// TIA Portal project "Pompe_4" (V15.1)

(* hardware
DEVICE "S71500/ET200MP station_1"  S7-1500 station
   slot 0: "Rail_0"  Rack  6ES7 590-1***0-0AA0
   slot 1: "PLC_1"  CPU 1513-1 PN  6ES7 513-1AL02-0AB0  V2.6
      slot 3: "CPU display_1"  6ES7591-1AA00-0AA0
DEVICE "HMI_1"  KTP900 Basic PN
   slot 0: "HMI_1"  KTP900 Basic PN  6AV2 123-2JB03-0AX0  15.1.0.0
   slot 1: "HMI_RT_1"  KTP900 Basic PN  6AV2 123-2JB03-0AX0  15.1.0.0
   slot 5: "HMI_1.IE_CP_1"  PROFINET Interface  15.0.1.0
      slot 1: "PROFINET Interface_1"  PROFINET Interface
         slot 1: "Port_1"  Port
*)

// ===== PLC "PLC_1"  CPU 1513-1 PN =====

VAR_GLOBAL   // PLC tag table "Default tag table"
   "Clock_Byte" AT %MB0 : Byte;
   "Clock_10Hz" AT %M0.0 : Bool;
   "Clock_5Hz" AT %M0.1 : Bool;
   "Clock_2.5Hz" AT %M0.2 : Bool;
   "Clock_2Hz" AT %M0.3 : Bool;
   "Clock_1.25Hz" AT %M0.4 : Bool;
   "Clock_1Hz" AT %M0.5 : Bool;
   "Clock_0.625Hz" AT %M0.6 : Bool;
   "Clock_0.5Hz" AT %M0.7 : Bool;
END_VAR

TYPE "typeLogEntry"
   STRUCT
      Timestamp : DTL;
      Level : Real;
      Mode : DInt;
      ESD_Active : Bool;
      Fault_Active : Bool;
   END_STRUCT;
END_TYPE

// folder: Alarme/Avarii

DATA_BLOCK "Alarme_DB"   // DB1
{ S7_Optimized_Access := 'TRUE' }
VERSION : 0.1
   VAR
      gather : Word;
      "array" : Array[0..15] of Bool;
   END_VAR
BEGIN
END_DATA_BLOCK

DATA_BLOCK "Avarii_DB"   // DB2
{ S7_Optimized_Access := 'TRUE' }
VERSION : 0.1
   VAR
      esd_1 : Bool;
      btn_esd_1 : Bool;
      reset_esd_1 : Bool;
      avarie_sistem_1 : Bool;
      btn_avarie_sistem_1 : Bool;
      reset_avarie_sistem_1 : Bool;
      esd_2 : Bool;
      btn_esd_2 : Bool;
      reset_esd_2 : Bool;
      avarie_sistem_2 : Bool;
      btn_avarie_sistem_2 : Bool;
      reset_avarie_sistem_2 : Bool;
      esd_3 : Bool;
      btn_esd_3 : Bool;
      reset_esd_3 : Bool;
      avarie_sistem_3 : Bool;
      btn_avarie_sistem_3 : Bool;
      reset_avarie_sistem_3 : Bool;
      esd_4 : Bool;
      btn_esd_4 : Bool;
      reset_esd_4 : Bool;
      avarie_sistem_4 : Bool;
      btn_avarie_sistem_4 : Bool;
      reset_avarie_sistem_4 : Bool;
   END_VAR
BEGIN
END_DATA_BLOCK

// folder: DB-Functii-Networks

DATA_BLOCK "Sistem_2"   // DB13
{ S7_Optimized_Access := 'TRUE' }
VERSION : 0.1
// stored: InstanceOfName Sistem
"Sistem"
BEGIN
END_DATA_BLOCK

DATA_BLOCK "Sistem_1"   // DB15
{ S7_Optimized_Access := 'TRUE' }
VERSION : 0.1
// stored: InstanceOfName Sistem
"Sistem"
BEGIN
END_DATA_BLOCK

DATA_BLOCK "Sistem_3"   // DB16
{ S7_Optimized_Access := 'TRUE' }
VERSION : 0.1
// stored: InstanceOfName Sistem
"Sistem"
BEGIN
END_DATA_BLOCK

DATA_BLOCK "Sistem_4"   // DB17
{ S7_Optimized_Access := 'TRUE' }
VERSION : 0.1
// stored: InstanceOfName Sistem
"Sistem"
BEGIN
END_DATA_BLOCK

DATA_BLOCK "Logs_DB_1"   // DB21
{ S7_Optimized_Access := 'TRUE' }
VERSION : 0.1
// stored: InstanceOfName Logs
"Logs"
BEGIN
END_DATA_BLOCK

DATA_BLOCK "Logs_DB_2"   // DB22
{ S7_Optimized_Access := 'TRUE' }
VERSION : 0.1
// stored: InstanceOfName Logs
"Logs"
BEGIN
END_DATA_BLOCK

DATA_BLOCK "Logs_DB_3"   // DB23
{ S7_Optimized_Access := 'TRUE' }
VERSION : 0.1
// stored: InstanceOfName Logs
"Logs"
BEGIN
END_DATA_BLOCK

DATA_BLOCK "Logs_DB_4"   // DB24
{ S7_Optimized_Access := 'TRUE' }
VERSION : 0.1
// stored: InstanceOfName Logs
"Logs"
BEGIN
END_DATA_BLOCK

// folder: DB-Functii-Networks/DB-Functii-Sistem

DATA_BLOCK "Pompa_sistem_1"   // DB8
{ S7_Optimized_Access := 'TRUE' }
VERSION : 0.1
// stored: InstanceOfName Pompa
"Pompa"
BEGIN
END_DATA_BLOCK

DATA_BLOCK "Vana_sistem_1"   // DB9
{ S7_Optimized_Access := 'TRUE' }
VERSION : 0.1
// stored: InstanceOfName Vana
"Vana"
BEGIN
END_DATA_BLOCK

DATA_BLOCK "Simulare_sistem_1"   // DB14
{ S7_Optimized_Access := 'TRUE' }
VERSION : 0.1
// stored: InstanceOfName Simulare
"Simulare"
BEGIN
END_DATA_BLOCK

// folder: Logs

DATA_BLOCK "Logs1_DB"   // DB7
{ S7_Optimized_Access := 'TRUE' }
VERSION : 0.1
   VAR
      Log_Array : Array[0..100] of "typeLogEntry";
      index : Int;
      index_write : Int;
      target_index : Int;
      btn_jump : Bool;
      btn_prev : Bool;
      btn_next : Bool;
      btn_latest : Bool;
      Display_Entry : "typeLogEntry";
   END_VAR
BEGIN
END_DATA_BLOCK

DATA_BLOCK "Logs2_DB"   // DB25
{ S7_Optimized_Access := 'TRUE' }
VERSION : 0.1
   VAR
      Log_Array : Array[0..100] of "typeLogEntry";
      index : Int;
      index_write : Int;
      target_index : Int;
      btn_jump : Bool;
      btn_prev : Bool;
      btn_next : Bool;
      btn_latest : Bool;
      Display_Entry : "typeLogEntry";
   END_VAR
BEGIN
END_DATA_BLOCK

DATA_BLOCK "Logs3_DB"   // DB26
{ S7_Optimized_Access := 'TRUE' }
VERSION : 0.1
   VAR
      Log_Array : Array[0..100] of "typeLogEntry";
      index : Int;
      index_write : Int;
      target_index : Int;
      btn_jump : Bool;
      btn_prev : Bool;
      btn_next : Bool;
      btn_latest : Bool;
      Display_Entry : "typeLogEntry";
   END_VAR
BEGIN
END_DATA_BLOCK

DATA_BLOCK "Logs4_DB"   // DB27
{ S7_Optimized_Access := 'TRUE' }
VERSION : 0.1
   VAR
      Log_Array : Array[0..100] of "typeLogEntry";
      index : Int;
      index_write : Int;
      target_index : Int;
      btn_jump : Bool;
      btn_prev : Bool;
      btn_next : Bool;
      btn_latest : Bool;
      Display_Entry : "typeLogEntry";
   END_VAR
BEGIN
END_DATA_BLOCK

// folder: Sisteme_DB

DATA_BLOCK "Sistem_1_DB"   // DB3
{ S7_Optimized_Access := 'TRUE' }
VERSION : 0.1
   VAR
      nivel_maxim : Real := 100.0;
      debit_vana : Real := 2.5;
      debit_pompa : Real := 2.5;
      comanda_pornire_pompa : Bool;
      comanda_pornire_vana : Bool;
      pornire_pompa_pid : Bool;
      pornire_vana_pid : Bool;
      permisiune_start : Bool;
      setpoint_pid : Real;
      nivel_bazin : Real;
      pid_output : Real;
      btn_start : Bool;
      btn_stop : Bool;
      plecare_pompa : Bool;
      plecare_vana : Bool;
      indicator_pornit : Bool;
      "mod" : DInt;
   END_VAR
BEGIN
END_DATA_BLOCK

DATA_BLOCK "Sistem_2_DB"   // DB4
{ S7_Optimized_Access := 'TRUE' }
VERSION : 0.1
   VAR
      nivel_maxim : Real := 100.0;
      debit_vana : Real := 3.4;
      debit_pompa : Real := 1.3;
      comanda_pornire_pompa : Bool;
      comanda_pornire_vana : Bool;
      pornire_pompa_pid : Bool;
      pornire_vana_pid : Bool;
      permisiune_start : Bool;
      setpoint_pid : Real;
      nivel_bazin : Real;
      pid_output : Real;
      btn_start : Bool;
      btn_stop : Bool;
      plecare_pompa : Bool;
      plecare_vana : Bool;
      indicator_pornit : Bool;
      "mod" : DInt;
   END_VAR
BEGIN
END_DATA_BLOCK

DATA_BLOCK "Sistem_3_DB"   // DB5
{ S7_Optimized_Access := 'TRUE' }
VERSION : 0.1
   VAR
      nivel_maxim : Real := 100.0;
      debit_vana : Real := 5.7;
      debit_pompa : Real := 1.2;
      comanda_pornire_pompa : Bool;
      comanda_pornire_vana : Bool;
      pornire_pompa_pid : Bool;
      pornire_vana_pid : Bool;
      permisiune_start : Bool;
      setpoint_pid : Real;
      nivel_bazin : Real;
      pid_output : Real;
      btn_start : Bool;
      btn_stop : Bool;
      plecare_pompa : Bool;
      plecare_vana : Bool;
      indicator_pornit : Bool;
      "mod" : DInt;
   END_VAR
BEGIN
END_DATA_BLOCK

DATA_BLOCK "Sistem_4_DB"   // DB6
{ S7_Optimized_Access := 'TRUE' }
VERSION : 0.1
   VAR
      nivel_maxim : Real := 100.0;
      debit_vana : Real := 1.8;
      debit_pompa : Real := 3.6;
      comanda_pornire_pompa : Bool;
      comanda_pornire_vana : Bool;
      pornire_pompa_pid : Bool;
      pornire_vana_pid : Bool;
      permisiune_start : Bool;
      setpoint_pid : Real;
      nivel_bazin : Real;
      pid_output : Real;
      btn_start : Bool;
      btn_stop : Bool;
      plecare_pompa : Bool;
      plecare_vana : Bool;
      indicator_pornit : Bool;
      "mod" : DInt;
   END_VAR
BEGIN
END_DATA_BLOCK

// folder: System blocks/Program resources

DATA_BLOCK "timer_reset_pornire_vana"   // DB10
{ S7_Optimized_Access := 'TRUE' }
AUTHOR : Simatic
FAMILY : IEC
NAME : IEC_TMR
VERSION : 1.0
// stored: InstanceOfName IEC_TIMER
"IEC_TIMER"
BEGIN
END_DATA_BLOCK

DATA_BLOCK "timer_reset_pornire_pompa"   // DB11
{ S7_Optimized_Access := 'TRUE' }
AUTHOR : Simatic
FAMILY : IEC
NAME : IEC_TMR
VERSION : 1.0
// stored: InstanceOfName IEC_TIMER
"IEC_TIMER"
BEGIN
END_DATA_BLOCK

// folder: (top level)

ORGANIZATION_BLOCK "Main"   // OB1, LAD, ProgramCycle
TITLE = "Main Program Sweep (Cycle)"
{ S7_Optimized_Access := 'TRUE' }
VERSION : 0.1
   VAR_INPUT
      Initial_Call : Bool;   // Initial call of this OB
      Remanence : Bool;   // =True, if remanent data are available
   END_VAR
BEGIN

REGION Network 1: Gather pe alarme
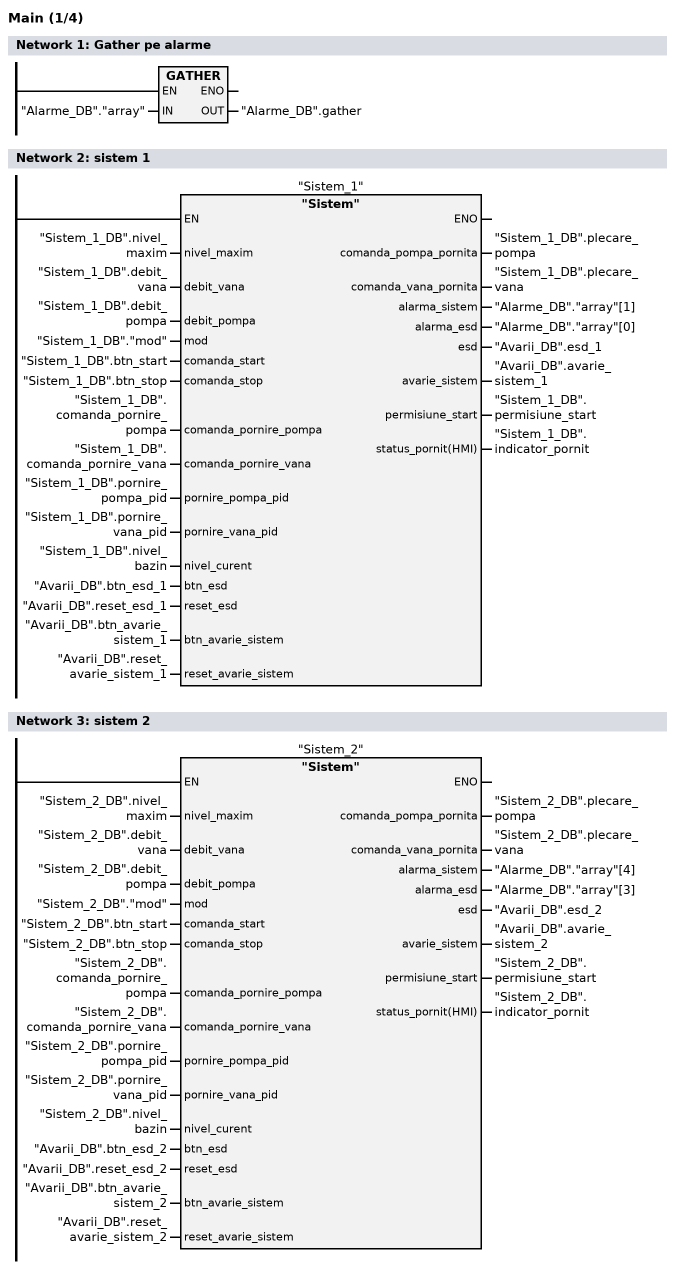
   GATHER(IN := "Alarme_DB"."array", OUT => "Alarme_DB".gather);
END_REGION

REGION Network 2: sistem 1
   RUNG wire#powerrail
      "Sistem_1"(nivel_maxim := "Sistem_1_DB".nivel_maxim, debit_vana := "Sistem_1_DB".debit_vana, debit_pompa := "Sistem_1_DB".debit_pompa, "mod" := "Sistem_1_DB"."mod", comanda_start := "Sistem_1_DB".btn_start, comanda_stop := "Sistem_1_DB".btn_stop, comanda_pornire_pompa := "Sistem_1_DB".comanda_pornire_pompa, comanda_pornire_vana := "Sistem_1_DB".comanda_pornire_vana, pornire_pompa_pid := "Sistem_1_DB".pornire_pompa_pid, pornire_vana_pid := "Sistem_1_DB".pornire_vana_pid, nivel_curent := "Sistem_1_DB".nivel_bazin, btn_esd := "Avarii_DB".btn_esd_1, reset_esd := "Avarii_DB".reset_esd_1, btn_avarie_sistem := "Avarii_DB".btn_avarie_sistem_1, reset_avarie_sistem := "Avarii_DB".reset_avarie_sistem_1, comanda_pompa_pornita => "Sistem_1_DB".plecare_pompa, comanda_vana_pornita => "Sistem_1_DB".plecare_vana, alarma_sistem => "Alarme_DB"."array"[1], alarma_esd => "Alarme_DB"."array"[0], esd => "Avarii_DB".esd_1, avarie_sistem => "Avarii_DB".avarie_sistem_1, permisiune_start => "Sistem_1_DB".permisiune_start, "status_pornit(HMI)" => "Sistem_1_DB".indicator_pornit)
   END_RUNG
   // the same network as SCL:
   "Sistem_1"(nivel_maxim := "Sistem_1_DB".nivel_maxim,   // "Sistem"
              debit_vana := "Sistem_1_DB".debit_vana,
              debit_pompa := "Sistem_1_DB".debit_pompa,
              "mod" := "Sistem_1_DB"."mod",
              comanda_start := "Sistem_1_DB".btn_start,
              comanda_stop := "Sistem_1_DB".btn_stop,
              comanda_pornire_pompa := "Sistem_1_DB".comanda_pornire_pompa,
              comanda_pornire_vana := "Sistem_1_DB".comanda_pornire_vana,
              pornire_pompa_pid := "Sistem_1_DB".pornire_pompa_pid,
              pornire_vana_pid := "Sistem_1_DB".pornire_vana_pid,
              nivel_curent := "Sistem_1_DB".nivel_bazin,
              btn_esd := "Avarii_DB".btn_esd_1,
              reset_esd := "Avarii_DB".reset_esd_1,
              btn_avarie_sistem := "Avarii_DB".btn_avarie_sistem_1,
              reset_avarie_sistem := "Avarii_DB".reset_avarie_sistem_1,
              comanda_pompa_pornita => "Sistem_1_DB".plecare_pompa,
              comanda_vana_pornita => "Sistem_1_DB".plecare_vana,
              alarma_sistem => "Alarme_DB"."array"[1],
              alarma_esd => "Alarme_DB"."array"[0],
              esd => "Avarii_DB".esd_1,
              avarie_sistem => "Avarii_DB".avarie_sistem_1,
              permisiune_start => "Sistem_1_DB".permisiune_start,
              "status_pornit(HMI)" => "Sistem_1_DB".indicator_pornit);
END_REGION

REGION Network 3: sistem 2
   RUNG wire#powerrail
      "Sistem_2"(nivel_maxim := "Sistem_2_DB".nivel_maxim, debit_vana := "Sistem_2_DB".debit_vana, debit_pompa := "Sistem_2_DB".debit_pompa, "mod" := "Sistem_2_DB"."mod", comanda_start := "Sistem_2_DB".btn_start, comanda_stop := "Sistem_2_DB".btn_stop, comanda_pornire_pompa := "Sistem_2_DB".comanda_pornire_pompa, comanda_pornire_vana := "Sistem_2_DB".comanda_pornire_vana, pornire_pompa_pid := "Sistem_2_DB".pornire_pompa_pid, pornire_vana_pid := "Sistem_2_DB".pornire_vana_pid, nivel_curent := "Sistem_2_DB".nivel_bazin, btn_esd := "Avarii_DB".btn_esd_2, reset_esd := "Avarii_DB".reset_esd_2, btn_avarie_sistem := "Avarii_DB".btn_avarie_sistem_2, reset_avarie_sistem := "Avarii_DB".reset_avarie_sistem_2, comanda_pompa_pornita => "Sistem_2_DB".plecare_pompa, comanda_vana_pornita => "Sistem_2_DB".plecare_vana, alarma_sistem => "Alarme_DB"."array"[4], alarma_esd => "Alarme_DB"."array"[3], esd => "Avarii_DB".esd_2, avarie_sistem => "Avarii_DB".avarie_sistem_2, permisiune_start => "Sistem_2_DB".permisiune_start, "status_pornit(HMI)" => "Sistem_2_DB".indicator_pornit)
   END_RUNG
   // the same network as SCL:
   "Sistem_2"(nivel_maxim := "Sistem_2_DB".nivel_maxim,   // "Sistem"
              debit_vana := "Sistem_2_DB".debit_vana,
              debit_pompa := "Sistem_2_DB".debit_pompa,
              "mod" := "Sistem_2_DB"."mod",
              comanda_start := "Sistem_2_DB".btn_start,
              comanda_stop := "Sistem_2_DB".btn_stop,
              comanda_pornire_pompa := "Sistem_2_DB".comanda_pornire_pompa,
              comanda_pornire_vana := "Sistem_2_DB".comanda_pornire_vana,
              pornire_pompa_pid := "Sistem_2_DB".pornire_pompa_pid,
              pornire_vana_pid := "Sistem_2_DB".pornire_vana_pid,
              nivel_curent := "Sistem_2_DB".nivel_bazin,
              btn_esd := "Avarii_DB".btn_esd_2,
              reset_esd := "Avarii_DB".reset_esd_2,
              btn_avarie_sistem := "Avarii_DB".btn_avarie_sistem_2,
              reset_avarie_sistem := "Avarii_DB".reset_avarie_sistem_2,
              comanda_pompa_pornita => "Sistem_2_DB".plecare_pompa,
              comanda_vana_pornita => "Sistem_2_DB".plecare_vana,
              alarma_sistem => "Alarme_DB"."array"[4],
              alarma_esd => "Alarme_DB"."array"[3],
              esd => "Avarii_DB".esd_2,
              avarie_sistem => "Avarii_DB".avarie_sistem_2,
              permisiune_start => "Sistem_2_DB".permisiune_start,
              "status_pornit(HMI)" => "Sistem_2_DB".indicator_pornit);
END_REGION

REGION Network 4: sistem 3
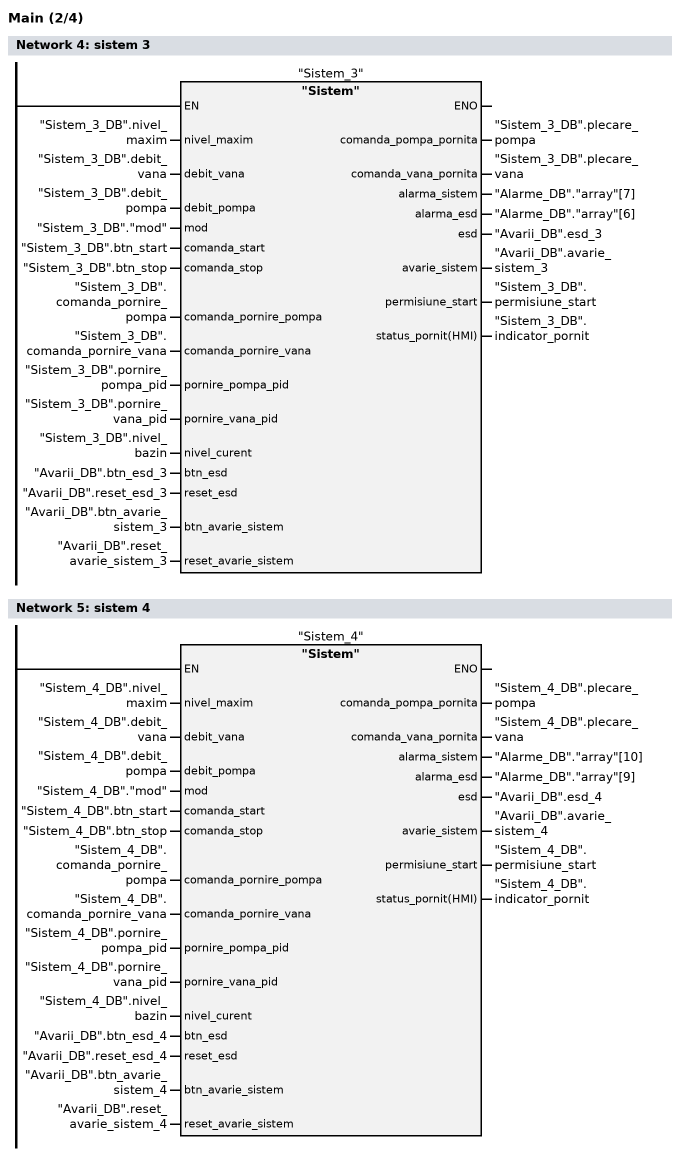
   RUNG wire#powerrail
      "Sistem_3"(nivel_maxim := "Sistem_3_DB".nivel_maxim, debit_vana := "Sistem_3_DB".debit_vana, debit_pompa := "Sistem_3_DB".debit_pompa, "mod" := "Sistem_3_DB"."mod", comanda_start := "Sistem_3_DB".btn_start, comanda_stop := "Sistem_3_DB".btn_stop, comanda_pornire_pompa := "Sistem_3_DB".comanda_pornire_pompa, comanda_pornire_vana := "Sistem_3_DB".comanda_pornire_vana, pornire_pompa_pid := "Sistem_3_DB".pornire_pompa_pid, pornire_vana_pid := "Sistem_3_DB".pornire_vana_pid, nivel_curent := "Sistem_3_DB".nivel_bazin, btn_esd := "Avarii_DB".btn_esd_3, reset_esd := "Avarii_DB".reset_esd_3, btn_avarie_sistem := "Avarii_DB".btn_avarie_sistem_3, reset_avarie_sistem := "Avarii_DB".reset_avarie_sistem_3, comanda_pompa_pornita => "Sistem_3_DB".plecare_pompa, comanda_vana_pornita => "Sistem_3_DB".plecare_vana, alarma_sistem => "Alarme_DB"."array"[7], alarma_esd => "Alarme_DB"."array"[6], esd => "Avarii_DB".esd_3, avarie_sistem => "Avarii_DB".avarie_sistem_3, permisiune_start => "Sistem_3_DB".permisiune_start, "status_pornit(HMI)" => "Sistem_3_DB".indicator_pornit)
   END_RUNG
   // the same network as SCL:
   "Sistem_3"(nivel_maxim := "Sistem_3_DB".nivel_maxim,   // "Sistem"
              debit_vana := "Sistem_3_DB".debit_vana,
              debit_pompa := "Sistem_3_DB".debit_pompa,
              "mod" := "Sistem_3_DB"."mod",
              comanda_start := "Sistem_3_DB".btn_start,
              comanda_stop := "Sistem_3_DB".btn_stop,
              comanda_pornire_pompa := "Sistem_3_DB".comanda_pornire_pompa,
              comanda_pornire_vana := "Sistem_3_DB".comanda_pornire_vana,
              pornire_pompa_pid := "Sistem_3_DB".pornire_pompa_pid,
              pornire_vana_pid := "Sistem_3_DB".pornire_vana_pid,
              nivel_curent := "Sistem_3_DB".nivel_bazin,
              btn_esd := "Avarii_DB".btn_esd_3,
              reset_esd := "Avarii_DB".reset_esd_3,
              btn_avarie_sistem := "Avarii_DB".btn_avarie_sistem_3,
              reset_avarie_sistem := "Avarii_DB".reset_avarie_sistem_3,
              comanda_pompa_pornita => "Sistem_3_DB".plecare_pompa,
              comanda_vana_pornita => "Sistem_3_DB".plecare_vana,
              alarma_sistem => "Alarme_DB"."array"[7],
              alarma_esd => "Alarme_DB"."array"[6],
              esd => "Avarii_DB".esd_3,
              avarie_sistem => "Avarii_DB".avarie_sistem_3,
              permisiune_start => "Sistem_3_DB".permisiune_start,
              "status_pornit(HMI)" => "Sistem_3_DB".indicator_pornit);
END_REGION

REGION Network 5: sistem 4
   RUNG wire#powerrail
      "Sistem_4"(nivel_maxim := "Sistem_4_DB".nivel_maxim, debit_vana := "Sistem_4_DB".debit_vana, debit_pompa := "Sistem_4_DB".debit_pompa, "mod" := "Sistem_4_DB"."mod", comanda_start := "Sistem_4_DB".btn_start, comanda_stop := "Sistem_4_DB".btn_stop, comanda_pornire_pompa := "Sistem_4_DB".comanda_pornire_pompa, comanda_pornire_vana := "Sistem_4_DB".comanda_pornire_vana, pornire_pompa_pid := "Sistem_4_DB".pornire_pompa_pid, pornire_vana_pid := "Sistem_4_DB".pornire_vana_pid, nivel_curent := "Sistem_4_DB".nivel_bazin, btn_esd := "Avarii_DB".btn_esd_4, reset_esd := "Avarii_DB".reset_esd_4, btn_avarie_sistem := "Avarii_DB".btn_avarie_sistem_4, reset_avarie_sistem := "Avarii_DB".reset_avarie_sistem_4, comanda_pompa_pornita => "Sistem_4_DB".plecare_pompa, comanda_vana_pornita => "Sistem_4_DB".plecare_vana, alarma_sistem => "Alarme_DB"."array"[10], alarma_esd => "Alarme_DB"."array"[9], esd => "Avarii_DB".esd_4, avarie_sistem => "Avarii_DB".avarie_sistem_4, permisiune_start => "Sistem_4_DB".permisiune_start, "status_pornit(HMI)" => "Sistem_4_DB".indicator_pornit)
   END_RUNG
   // the same network as SCL:
   "Sistem_4"(nivel_maxim := "Sistem_4_DB".nivel_maxim,   // "Sistem"
              debit_vana := "Sistem_4_DB".debit_vana,
              debit_pompa := "Sistem_4_DB".debit_pompa,
              "mod" := "Sistem_4_DB"."mod",
              comanda_start := "Sistem_4_DB".btn_start,
              comanda_stop := "Sistem_4_DB".btn_stop,
              comanda_pornire_pompa := "Sistem_4_DB".comanda_pornire_pompa,
              comanda_pornire_vana := "Sistem_4_DB".comanda_pornire_vana,
              pornire_pompa_pid := "Sistem_4_DB".pornire_pompa_pid,
              pornire_vana_pid := "Sistem_4_DB".pornire_vana_pid,
              nivel_curent := "Sistem_4_DB".nivel_bazin,
              btn_esd := "Avarii_DB".btn_esd_4,
              reset_esd := "Avarii_DB".reset_esd_4,
              btn_avarie_sistem := "Avarii_DB".btn_avarie_sistem_4,
              reset_avarie_sistem := "Avarii_DB".reset_avarie_sistem_4,
              comanda_pompa_pornita => "Sistem_4_DB".plecare_pompa,
              comanda_vana_pornita => "Sistem_4_DB".plecare_vana,
              alarma_sistem => "Alarme_DB"."array"[10],
              alarma_esd => "Alarme_DB"."array"[9],
              esd => "Avarii_DB".esd_4,
              avarie_sistem => "Avarii_DB".avarie_sistem_4,
              permisiune_start => "Sistem_4_DB".permisiune_start,
              "status_pornit(HMI)" => "Sistem_4_DB".indicator_pornit);
END_REGION

REGION Network 6: logs 1
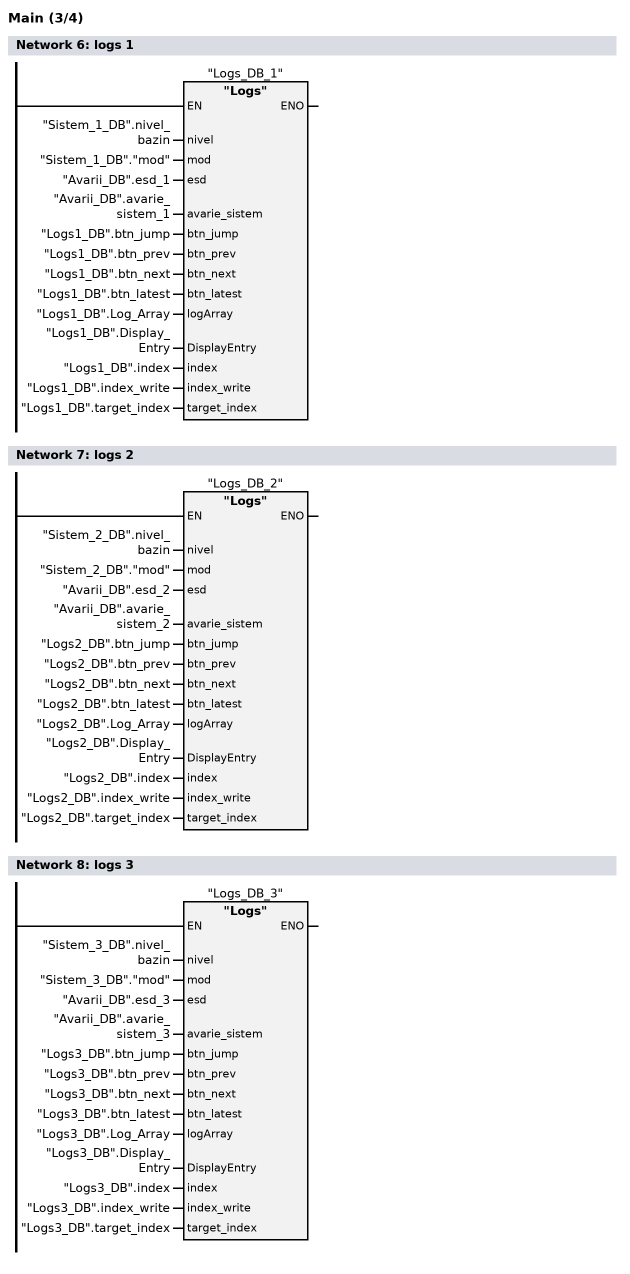
   RUNG wire#powerrail
      "Logs_DB_1"(nivel := "Sistem_1_DB".nivel_bazin, "mod" := "Sistem_1_DB"."mod", esd := "Avarii_DB".esd_1, avarie_sistem := "Avarii_DB".avarie_sistem_1, btn_jump := "Logs1_DB".btn_jump, btn_prev := "Logs1_DB".btn_prev, btn_next := "Logs1_DB".btn_next, btn_latest := "Logs1_DB".btn_latest, logArray := "Logs1_DB".Log_Array, DisplayEntry := "Logs1_DB".Display_Entry, index := "Logs1_DB".index, index_write := "Logs1_DB".index_write, target_index := "Logs1_DB".target_index)
   END_RUNG
   // the same network as SCL:
   "Logs_DB_1"(nivel := "Sistem_1_DB".nivel_bazin,   // "Logs"
               "mod" := "Sistem_1_DB"."mod",
               esd := "Avarii_DB".esd_1,
               avarie_sistem := "Avarii_DB".avarie_sistem_1,
               btn_jump := "Logs1_DB".btn_jump,
               btn_prev := "Logs1_DB".btn_prev,
               btn_next := "Logs1_DB".btn_next,
               btn_latest := "Logs1_DB".btn_latest,
               logArray := "Logs1_DB".Log_Array,
               DisplayEntry := "Logs1_DB".Display_Entry,
               index := "Logs1_DB".index,
               index_write := "Logs1_DB".index_write,
               target_index := "Logs1_DB".target_index);
END_REGION

REGION Network 7: logs 2
   RUNG wire#powerrail
      "Logs_DB_2"(nivel := "Sistem_2_DB".nivel_bazin, "mod" := "Sistem_2_DB"."mod", esd := "Avarii_DB".esd_2, avarie_sistem := "Avarii_DB".avarie_sistem_2, btn_jump := "Logs2_DB".btn_jump, btn_prev := "Logs2_DB".btn_prev, btn_next := "Logs2_DB".btn_next, btn_latest := "Logs2_DB".btn_latest, logArray := "Logs2_DB".Log_Array, DisplayEntry := "Logs2_DB".Display_Entry, index := "Logs2_DB".index, index_write := "Logs2_DB".index_write, target_index := "Logs2_DB".target_index)
   END_RUNG
   // the same network as SCL:
   "Logs_DB_2"(nivel := "Sistem_2_DB".nivel_bazin,   // "Logs"
               "mod" := "Sistem_2_DB"."mod",
               esd := "Avarii_DB".esd_2,
               avarie_sistem := "Avarii_DB".avarie_sistem_2,
               btn_jump := "Logs2_DB".btn_jump,
               btn_prev := "Logs2_DB".btn_prev,
               btn_next := "Logs2_DB".btn_next,
               btn_latest := "Logs2_DB".btn_latest,
               logArray := "Logs2_DB".Log_Array,
               DisplayEntry := "Logs2_DB".Display_Entry,
               index := "Logs2_DB".index,
               index_write := "Logs2_DB".index_write,
               target_index := "Logs2_DB".target_index);
END_REGION

REGION Network 8: logs 3
   RUNG wire#powerrail
      "Logs_DB_3"(nivel := "Sistem_3_DB".nivel_bazin, "mod" := "Sistem_3_DB"."mod", esd := "Avarii_DB".esd_3, avarie_sistem := "Avarii_DB".avarie_sistem_3, btn_jump := "Logs3_DB".btn_jump, btn_prev := "Logs3_DB".btn_prev, btn_next := "Logs3_DB".btn_next, btn_latest := "Logs3_DB".btn_latest, logArray := "Logs3_DB".Log_Array, DisplayEntry := "Logs3_DB".Display_Entry, index := "Logs3_DB".index, index_write := "Logs3_DB".index_write, target_index := "Logs3_DB".target_index)
   END_RUNG
   // the same network as SCL:
   "Logs_DB_3"(nivel := "Sistem_3_DB".nivel_bazin,   // "Logs"
               "mod" := "Sistem_3_DB"."mod",
               esd := "Avarii_DB".esd_3,
               avarie_sistem := "Avarii_DB".avarie_sistem_3,
               btn_jump := "Logs3_DB".btn_jump,
               btn_prev := "Logs3_DB".btn_prev,
               btn_next := "Logs3_DB".btn_next,
               btn_latest := "Logs3_DB".btn_latest,
               logArray := "Logs3_DB".Log_Array,
               DisplayEntry := "Logs3_DB".Display_Entry,
               index := "Logs3_DB".index,
               index_write := "Logs3_DB".index_write,
               target_index := "Logs3_DB".target_index);
END_REGION

REGION Network 9: logs 4
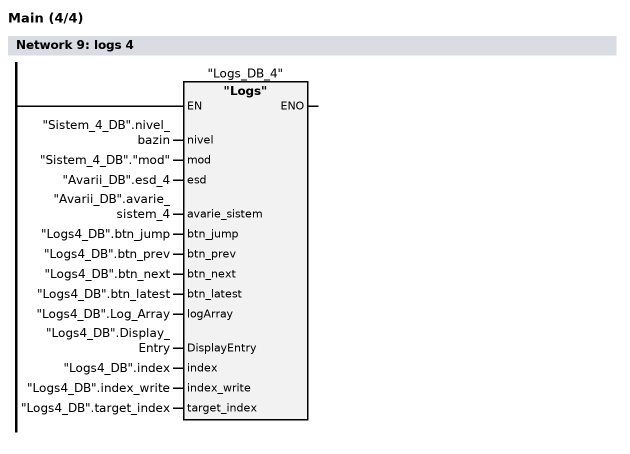
   RUNG wire#powerrail
      "Logs_DB_4"(nivel := "Sistem_4_DB".nivel_bazin, "mod" := "Sistem_4_DB"."mod", esd := "Avarii_DB".esd_4, avarie_sistem := "Avarii_DB".avarie_sistem_4, btn_jump := "Logs4_DB".btn_jump, btn_prev := "Logs4_DB".btn_prev, btn_next := "Logs4_DB".btn_next, btn_latest := "Logs4_DB".btn_latest, logArray := "Logs4_DB".Log_Array, DisplayEntry := "Logs4_DB".Display_Entry, index := "Logs4_DB".index, index_write := "Logs4_DB".index_write, target_index := "Logs4_DB".target_index)
   END_RUNG
   // the same network as SCL:
   "Logs_DB_4"(nivel := "Sistem_4_DB".nivel_bazin,   // "Logs"
               "mod" := "Sistem_4_DB"."mod",
               esd := "Avarii_DB".esd_4,
               avarie_sistem := "Avarii_DB".avarie_sistem_4,
               btn_jump := "Logs4_DB".btn_jump,
               btn_prev := "Logs4_DB".btn_prev,
               btn_next := "Logs4_DB".btn_next,
               btn_latest := "Logs4_DB".btn_latest,
               logArray := "Logs4_DB".Log_Array,
               DisplayEntry := "Logs4_DB".Display_Entry,
               index := "Logs4_DB".index,
               index_write := "Logs4_DB".index_write,
               target_index := "Logs4_DB".target_index);
END_REGION
END_ORGANIZATION_BLOCK

// folder: FB-Sistem

FUNCTION_BLOCK "Sistem"   // FB1, LAD
{ S7_Optimized_Access := 'TRUE' }
VERSION : 0.1
   VAR_INPUT
      nivel_maxim : Real;
      debit_vana : Real;
      debit_pompa : Real;
      "mod" : DInt;
   END_VAR
   VAR_OUTPUT
      comanda_pompa_pornita : Bool;
      comanda_vana_pornita : Bool;
      alarma_sistem : Bool;
      alarma_esd : Bool;
      esd : Bool;
      avarie_sistem : Bool;
      permisiune_start : Bool;
      "status_pornit(HMI)" : Bool;
   END_VAR
   VAR_IN_OUT
      comanda_start : Bool;
      comanda_stop : Bool;
      comanda_pornire_pompa : Bool;
      comanda_pornire_vana : Bool;
      pornire_pompa_pid : Bool;
      pornire_vana_pid : Bool;
      nivel_curent : Real;
      btn_esd : Bool;
      reset_esd : Bool;
      btn_avarie_sistem : Bool;
      reset_avarie_sistem : Bool;
   END_VAR
   VAR
      status_pornit_pompa : Bool;
      status_pornit_vana : Bool;
      resetare_comanda_vana : Bool;
      resetare_comanda_pompa : Bool;
      timer_reset_esd : TON_TIME;
      timer_reset_avarie_sistem : TON_TIME;
      timer_reset_comanda_stop : TON_TIME;
      Simulare_Instance : "Simulare";
      Vana_Instance : "Vana";
      Pompa_Instance : "Pompa";
   END_VAR
   VAR_TEMP   // added for the SCL form of the ladder/FBD networks
      _w1 : Bool;
      _w2 : Bool;
   END_VAR
BEGIN

REGION Network 1: comanda buton start
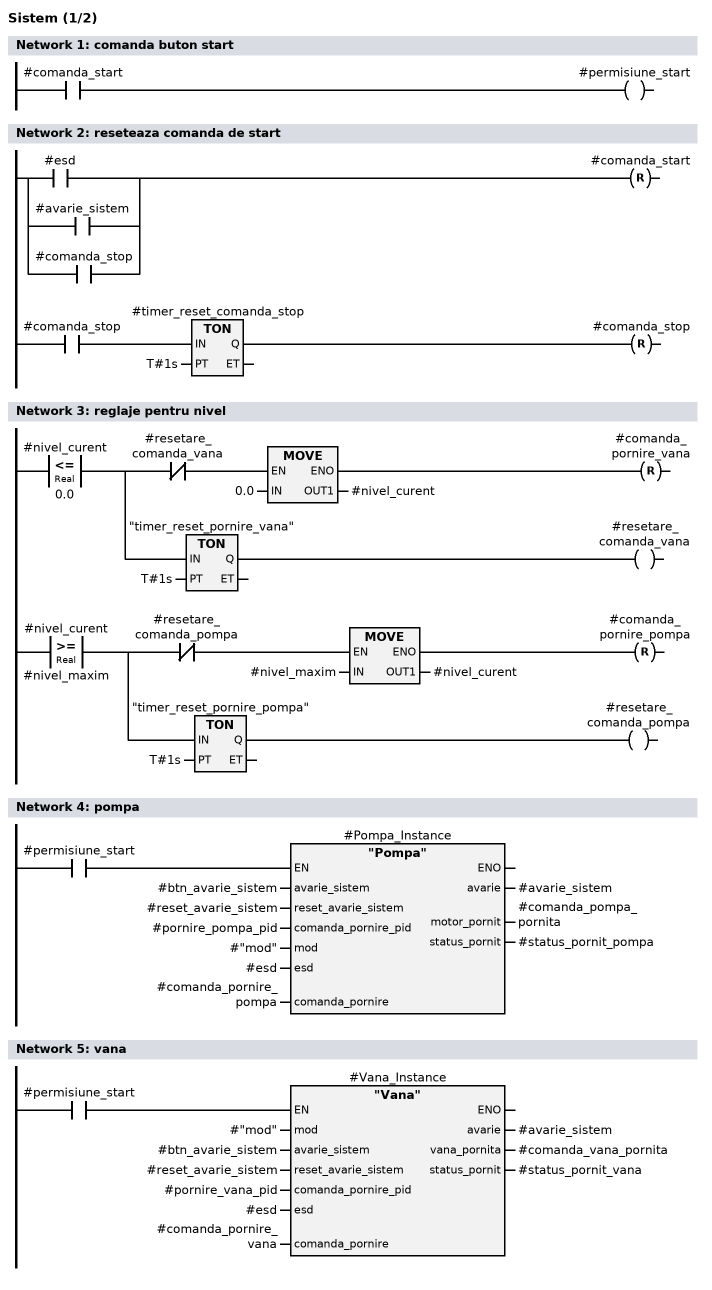
   RUNG wire#powerrail
      Contact( #comanda_start )
      Coil( #permisiune_start )
   END_RUNG
   // the same network as SCL:
   #permisiune_start := #comanda_start;
END_REGION

REGION Network 2: reseteaza comanda de start
   IF #esd OR #avarie_sistem OR #comanda_stop THEN #comanda_start := FALSE; END_IF;
   #timer_reset_comanda_stop(IN := #comanda_stop, PT := T#1s);   // TON
   IF #timer_reset_comanda_stop.Q THEN #comanda_stop := FALSE; END_IF;
END_REGION

REGION Network 3: reglaje pentru nivel
   #_w1 := #nivel_curent <= 0.0;
   IF #_w1 AND NOT #resetare_comanda_vana THEN
       #nivel_curent := 0.0;
       #comanda_pornire_vana := FALSE;
   END_IF;
   "timer_reset_pornire_vana".TON(IN := #_w1, PT := T#1s);
   #resetare_comanda_vana := "timer_reset_pornire_vana".Q;
   #_w2 := #nivel_curent >= #nivel_maxim;
   IF #_w2 AND NOT #resetare_comanda_pompa THEN
       #nivel_curent := #nivel_maxim;
       #comanda_pornire_pompa := FALSE;
   END_IF;
   "timer_reset_pornire_pompa".TON(IN := #_w2, PT := T#1s);
   #resetare_comanda_pompa := "timer_reset_pornire_pompa".Q;
END_REGION

REGION Network 4: pompa
   RUNG wire#powerrail
      Contact( #permisiune_start )
      #Pompa_Instance(avarie_sistem := #btn_avarie_sistem, reset_avarie_sistem := #reset_avarie_sistem, comanda_pornire_pid := #pornire_pompa_pid, "mod" := #"mod", esd := #esd, comanda_pornire := #comanda_pornire_pompa, avarie => #avarie_sistem, motor_pornit => #comanda_pompa_pornita, status_pornit => #status_pornit_pompa)
   END_RUNG
   // the same network as SCL:
   IF #permisiune_start THEN
       #Pompa_Instance(avarie_sistem := #btn_avarie_sistem,   // "Pompa"
                       reset_avarie_sistem := #reset_avarie_sistem,
                       comanda_pornire_pid := #pornire_pompa_pid,
                       "mod" := #"mod",
                       esd := #esd,
                       comanda_pornire := #comanda_pornire_pompa,
                       avarie => #avarie_sistem,
                       motor_pornit => #comanda_pompa_pornita,
                       status_pornit => #status_pornit_pompa);
   END_IF;
END_REGION

REGION Network 5: vana
   RUNG wire#powerrail
      Contact( #permisiune_start )
      #Vana_Instance("mod" := #"mod", avarie_sistem := #btn_avarie_sistem, reset_avarie_sistem := #reset_avarie_sistem, comanda_pornire_pid := #pornire_vana_pid, esd := #esd, comanda_pornire := #comanda_pornire_vana, avarie => #avarie_sistem, vana_pornita => #comanda_vana_pornita, status_pornit => #status_pornit_vana)
   END_RUNG
   // the same network as SCL:
   IF #permisiune_start THEN
       #Vana_Instance("mod" := #"mod",   // "Vana"
                      avarie_sistem := #btn_avarie_sistem,
                      reset_avarie_sistem := #reset_avarie_sistem,
                      comanda_pornire_pid := #pornire_vana_pid,
                      esd := #esd,
                      comanda_pornire := #comanda_pornire_vana,
                      avarie => #avarie_sistem,
                      vana_pornita => #comanda_vana_pornita,
                      status_pornit => #status_pornit_vana);
   END_IF;
END_REGION

REGION Network 6: status sistem pornit
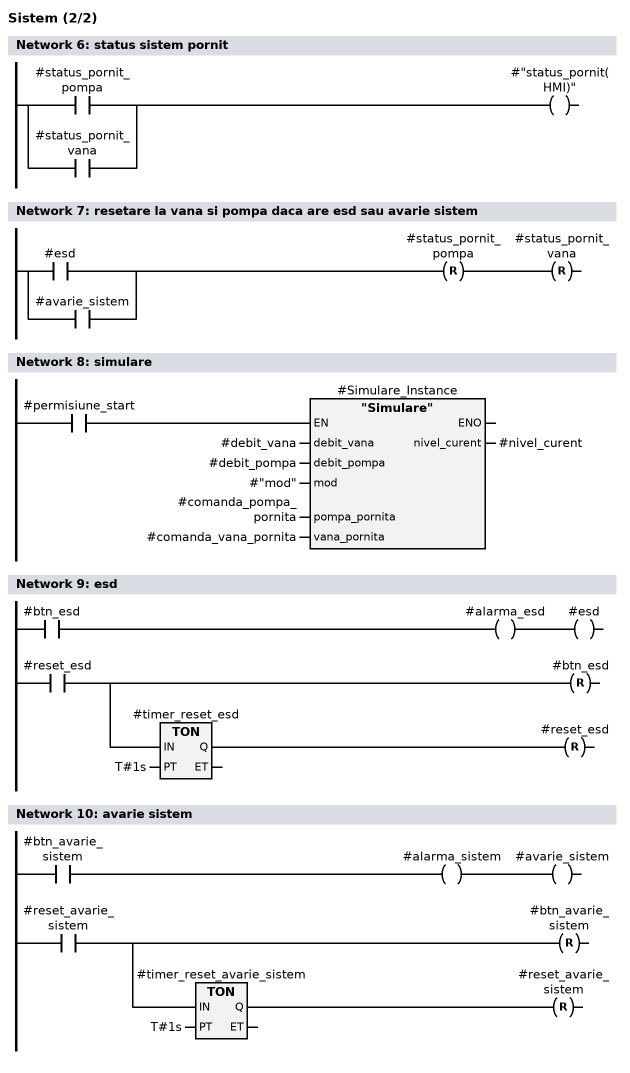
   RUNG wire#powerrail
      Contact( #status_pornit_pompa )
      wire#w1
      Coil( #"status_pornit(HMI)" )
   END_RUNG
   RUNG wire#powerrail
      Contact( #status_pornit_vana )
   END_RUNG wire#w1
   // the same network as SCL:
   #"status_pornit(HMI)" := #status_pornit_pompa OR #status_pornit_vana;
END_REGION

REGION Network 7: resetare la vana si pompa daca are esd sau avarie sistem
   RUNG wire#powerrail
      Contact( #esd )
      wire#w1
      R_Coil( #status_pornit_pompa )
      R_Coil( #status_pornit_vana )
   END_RUNG
   RUNG wire#powerrail
      Contact( #avarie_sistem )
   END_RUNG wire#w1
   // the same network as SCL:
   IF #esd OR #avarie_sistem THEN
       #status_pornit_pompa := FALSE;
       #status_pornit_vana := FALSE;
   END_IF;
END_REGION

REGION Network 8: simulare
   RUNG wire#powerrail
      Contact( #permisiune_start )
      #Simulare_Instance(debit_vana := #debit_vana, debit_pompa := #debit_pompa, "mod" := #"mod", pompa_pornita := #comanda_pompa_pornita, vana_pornita := #comanda_vana_pornita, nivel_curent => #nivel_curent)
   END_RUNG
   // the same network as SCL:
   IF #permisiune_start THEN
       #Simulare_Instance(debit_vana := #debit_vana,   // "Simulare"
                          debit_pompa := #debit_pompa,
                          "mod" := #"mod",
                          pompa_pornita := #comanda_pompa_pornita,
                          vana_pornita := #comanda_vana_pornita,
                          nivel_curent => #nivel_curent);
   END_IF;
END_REGION

REGION Network 9: esd
   #alarma_esd := #btn_esd;
   #esd := #btn_esd;
   IF #reset_esd THEN #btn_esd := FALSE; END_IF;
   #timer_reset_esd(IN := #reset_esd, PT := T#1s);   // TON
   IF #timer_reset_esd.Q THEN #reset_esd := FALSE; END_IF;
END_REGION

REGION Network 10: avarie sistem
   #alarma_sistem := #btn_avarie_sistem;
   #avarie_sistem := #btn_avarie_sistem;
   IF #reset_avarie_sistem THEN #btn_avarie_sistem := FALSE; END_IF;
   #timer_reset_avarie_sistem(IN := #reset_avarie_sistem, PT := T#1s);   // TON
   IF #timer_reset_avarie_sistem.Q THEN #reset_avarie_sistem := FALSE; END_IF;
END_REGION
END_FUNCTION_BLOCK

FUNCTION_BLOCK "Pompa"   // FB2, LAD
{ S7_Optimized_Access := 'TRUE' }
VERSION : 0.1
   VAR_INPUT
      avarie_sistem : Bool;
      reset_avarie_sistem : Bool;
      comanda_pornire_pid : Bool;
      "mod" : DInt;
      esd : Bool;
   END_VAR
   VAR_OUTPUT
      avarie : Bool;
      motor_pornit : Bool;
      status_pornit : Bool;
   END_VAR
   VAR_IN_OUT
      comanda_pornire : Bool;
   END_VAR
BEGIN

REGION Network 1: pornire pompa pe oricem od de functionare
   // 0 - manual, 1 - auto
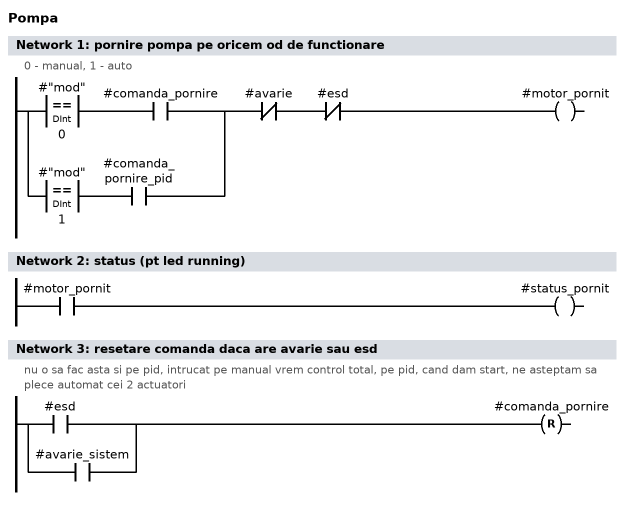
   RUNG wire#powerrail
      { S7_Templates := "SrcType := DInt" } EQ_Contact(in1 := #"mod", in2 := 0)
      Contact( #comanda_pornire )
      wire#w1
      I_Contact( #avarie )
      I_Contact( #esd )
      Coil( #motor_pornit )
   END_RUNG
   RUNG wire#powerrail
      { S7_Templates := "SrcType := DInt" } EQ_Contact(in1 := #"mod", in2 := 1)
      Contact( #comanda_pornire_pid )
   END_RUNG wire#w1
   // the same network as SCL:
   #motor_pornit := (((#"mod" = 0) AND #comanda_pornire) OR ((#"mod" = 1) AND #comanda_pornire_pid)) AND NOT #avarie AND NOT #esd;
END_REGION

REGION Network 2: status (pt led running)
   RUNG wire#powerrail
      Contact( #motor_pornit )
      Coil( #status_pornit )
   END_RUNG
   // the same network as SCL:
   #status_pornit := #motor_pornit;
END_REGION

REGION Network 3: resetare comanda daca are avarie sau esd
   // nu o sa fac asta si pe pid, intrucat pe manual vrem control total, pe pid, cand dam start, ne asteptam sa plece automat cei 2 actuatori
   RUNG wire#powerrail
      Contact( #esd )
      wire#w1
      R_Coil( #comanda_pornire )
   END_RUNG
   RUNG wire#powerrail
      Contact( #avarie_sistem )
   END_RUNG wire#w1
   // the same network as SCL:
   IF #esd OR #avarie_sistem THEN #comanda_pornire := FALSE; END_IF;
END_REGION
END_FUNCTION_BLOCK

FUNCTION_BLOCK "Vana"   // FB3, LAD
{ S7_Optimized_Access := 'TRUE' }
VERSION : 0.1
   VAR_INPUT
      "mod" : DInt;
      avarie_sistem : Bool;
      reset_avarie_sistem : Bool;
      comanda_pornire_pid : Bool;
      esd : Bool;
   END_VAR
   VAR_OUTPUT
      avarie : Bool;
      vana_pornita : Bool;
      status_pornit : Bool;
   END_VAR
   VAR_IN_OUT
      comanda_pornire : Bool;
   END_VAR
BEGIN

REGION Network 1: pornire pompa pe oricem od de functionare
   // 0 - manual, 1 - auto
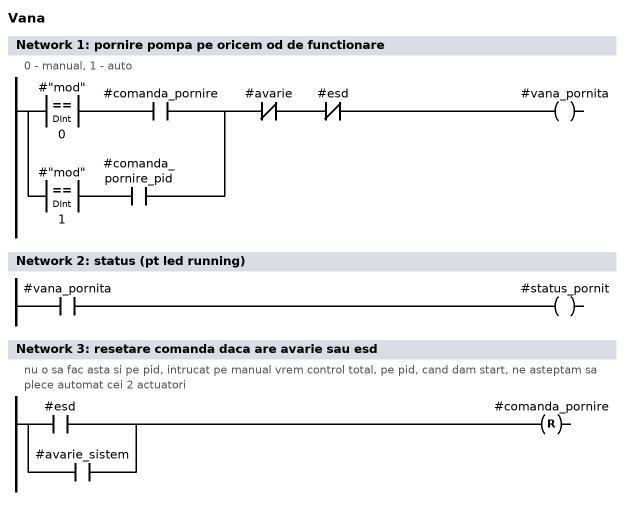
   RUNG wire#powerrail
      { S7_Templates := "SrcType := DInt" } EQ_Contact(in1 := #"mod", in2 := 0)
      Contact( #comanda_pornire )
      wire#w1
      I_Contact( #avarie )
      I_Contact( #esd )
      Coil( #vana_pornita )
   END_RUNG
   RUNG wire#powerrail
      { S7_Templates := "SrcType := DInt" } EQ_Contact(in1 := #"mod", in2 := 1)
      Contact( #comanda_pornire_pid )
   END_RUNG wire#w1
   // the same network as SCL:
   #vana_pornita := (((#"mod" = 0) AND #comanda_pornire) OR ((#"mod" = 1) AND #comanda_pornire_pid)) AND NOT #avarie AND NOT #esd;
END_REGION

REGION Network 2: status (pt led running)
   RUNG wire#powerrail
      Contact( #vana_pornita )
      Coil( #status_pornit )
   END_RUNG
   // the same network as SCL:
   #status_pornit := #vana_pornita;
END_REGION

REGION Network 3: resetare comanda daca are avarie sau esd
   // nu o sa fac asta si pe pid, intrucat pe manual vrem control total, pe pid, cand dam start, ne asteptam sa plece automat cei 2 actuatori
   RUNG wire#powerrail
      Contact( #esd )
      wire#w1
      R_Coil( #comanda_pornire )
   END_RUNG
   RUNG wire#powerrail
      Contact( #avarie_sistem )
   END_RUNG wire#w1
   // the same network as SCL:
   IF #esd OR #avarie_sistem THEN #comanda_pornire := FALSE; END_IF;
END_REGION
END_FUNCTION_BLOCK

FUNCTION_BLOCK "Simulare"   // FB4, LAD
{ S7_Optimized_Access := 'TRUE' }
VERSION : 0.1
   VAR_INPUT
      debit_vana : Real;
      debit_pompa : Real;
      "mod" : DInt;
      pompa_pornita : Bool;
      vana_pornita : Bool;
   END_VAR
   VAR_OUTPUT
      nivel_curent : Real;
   END_VAR
   VAR
      re1 : Bool;
      re2 : Bool;
   END_VAR
   VAR_TEMP   // added for the SCL form of the ladder/FBD networks
      _w1 : Bool;
   END_VAR
BEGIN

REGION Network 1: umple cu pompa
   // asta pe mod 0 manual, pe auto, o sa fie bloc separat cu pid
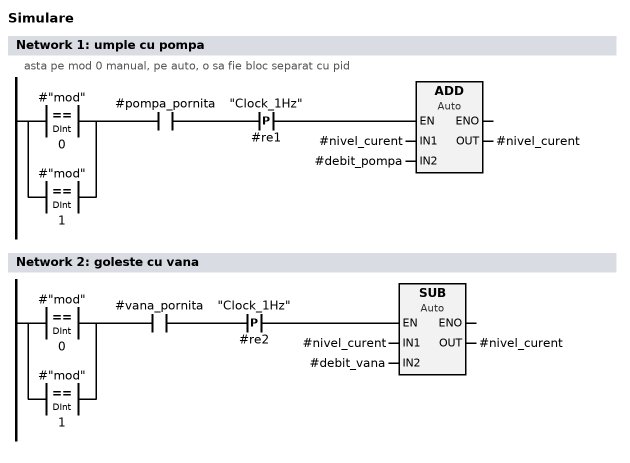
   RUNG wire#powerrail
      { S7_Templates := "SrcType := DInt" } EQ_Contact(in1 := #"mod", in2 := 0)
      wire#w1
      Contact( #pompa_pornita )
      P_Contact(operand := "Clock_1Hz", bit := #re1)
      Add(in1 := #nivel_curent, in2 := #debit_pompa, out => #nivel_curent)
   END_RUNG
   RUNG wire#powerrail
      { S7_Templates := "SrcType := DInt" } EQ_Contact(in1 := #"mod", in2 := 1)
   END_RUNG wire#w1
   // the same network as SCL:
   #_w1 := ((#"mod" = 0) OR (#"mod" = 1)) AND #pompa_pornita AND "Clock_1Hz" AND NOT #re1;   // rising edge of "Clock_1Hz"
   #re1 := "Clock_1Hz";
   IF #_w1 THEN #nivel_curent := #nivel_curent + #debit_pompa; END_IF;
END_REGION

REGION Network 2: goleste cu vana
   RUNG wire#powerrail
      { S7_Templates := "SrcType := DInt" } EQ_Contact(in1 := #"mod", in2 := 0)
      wire#w1
      Contact( #vana_pornita )
      P_Contact(operand := "Clock_1Hz", bit := #re2)
      Sub(in1 := #nivel_curent, in2 := #debit_vana, out => #nivel_curent)
   END_RUNG
   RUNG wire#powerrail
      { S7_Templates := "SrcType := DInt" } EQ_Contact(in1 := #"mod", in2 := 1)
   END_RUNG wire#w1
   // the same network as SCL:
   #_w1 := ((#"mod" = 0) OR (#"mod" = 1)) AND #vana_pornita AND "Clock_1Hz" AND NOT #re2;   // rising edge of "Clock_1Hz"
   #re2 := "Clock_1Hz";
   IF #_w1 THEN #nivel_curent := #nivel_curent - #debit_vana; END_IF;
END_REGION
END_FUNCTION_BLOCK

// folder: Logs

FUNCTION_BLOCK "Logs"   // FB5, LAD
{ S7_Optimized_Access := 'TRUE' }
VERSION : 0.1
   VAR_INPUT
      nivel : Real;
      "mod" : DInt;
      esd : Bool;
      avarie_sistem : Bool;
      btn_jump : Bool;
      btn_prev : Bool;
      btn_next : Bool;
      btn_latest : Bool;
   END_VAR
   VAR_IN_OUT
      logArray : Array[0..100] of "typeLogEntry";
      DisplayEntry : "typeLogEntry";
      index : Int;
      index_write : Int;
      target_index : Int;
   END_VAR
   VAR
      instLogTimer : TON_TIME;
      re1 : Bool;
      re2 : Bool;
      inc : Bool;
      dec : Bool;
      timerPulse : Bool;
   END_VAR
   VAR_TEMP
      statTimeError : Int;
   END_VAR
   VAR_TEMP   // added for the SCL form of the ladder/FBD networks
      _w1 : Bool;
   END_VAR
BEGIN

REGION Network 1 (SCL): retine valori in logs
   #instLogTimer(IN := NOT #timerPulse,
                 PT := T#3M);
   #timerPulse := #instLogTimer.Q;

   IF #timerPulse THEN
       IF #index_write < 1 OR #index_write > 100 THEN
           #index_write := 1;
       END_IF;

       #statTimeError := RD_SYS_T(#logArray[#index_write].Timestamp);
       #logArray[#index_write].Level := #nivel;
       #logArray[#index_write].Mode := #mod;
       #logArray[#index_write].ESD_Active := #esd;
       #logArray[#index_write].Fault_Active := #avarie_sistem;

       #index_write := #index_write + 1;
       IF #index_write > 100 THEN
           #index_write := 1;
       END_IF;
   END_IF;
END_REGION

REGION Network 2 (SCL): mergi la indexul cautat
   IF #btn_jump THEN
       #index := LIMIT(MN := 1, IN := #target_index, MX := 100);

   END_IF;
END_REGION

REGION Network 3: buton inainte
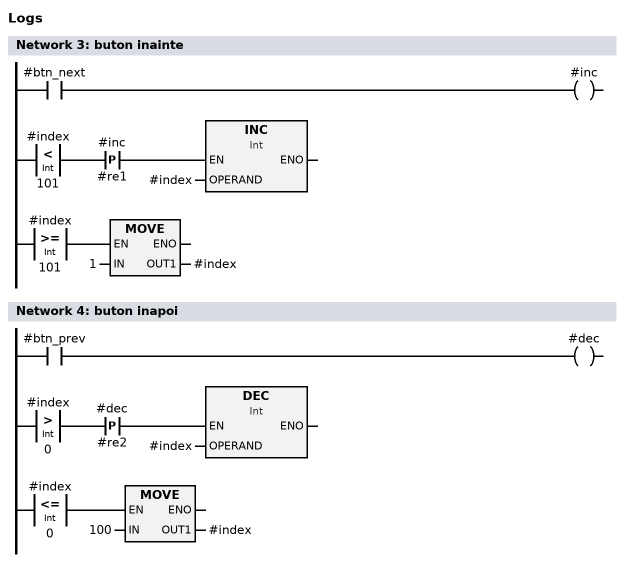
   RUNG wire#powerrail
      Contact( #btn_next )
      Coil( #inc )
   END_RUNG
   RUNG wire#powerrail
      { S7_Templates := "SrcType := Int" } LT_Contact(in1 := #index, in2 := 101)
      P_Contact(operand := #inc, bit := #re1)
      { S7_Templates := "DestType := Int" } Inc( #index )
   END_RUNG
   RUNG wire#powerrail
      { S7_Templates := "SrcType := Int" } GE_Contact(in1 := #index, in2 := 101)
      Move(in := 1, out1 => #index)
   END_RUNG
   // the same network as SCL:
   #inc := #btn_next;
   #_w1 := (#index < 101) AND #inc AND NOT #re1;   // rising edge of #inc
   #re1 := #inc;
   IF #_w1 THEN #index := #index + 1; END_IF;
   IF #index >= 101 THEN #index := 1; END_IF;
END_REGION

REGION Network 4: buton inapoi
   RUNG wire#powerrail
      Contact( #btn_prev )
      Coil( #dec )
   END_RUNG
   RUNG wire#powerrail
      { S7_Templates := "SrcType := Int" } GT_Contact(in1 := #index, in2 := 0)
      P_Contact(operand := #dec, bit := #re2)
      { S7_Templates := "DestType := Int" } Dec( #index )
   END_RUNG
   RUNG wire#powerrail
      { S7_Templates := "SrcType := Int" } LE_Contact(in1 := #index, in2 := 0)
      Move(in := 100, out1 => #index)
   END_RUNG
   // the same network as SCL:
   #dec := #btn_prev;
   #_w1 := (#index > 0) AND #dec AND NOT #re2;   // rising edge of #dec
   #re2 := #dec;
   IF #_w1 THEN #index := #index - 1; END_IF;
   IF #index <= 0 THEN #index := 100; END_IF;
END_REGION

REGION Network 5 (SCL): update pt indexul de pe hmi
   #DisplayEntry := #logArray[#index];
END_REGION

REGION Network 6 (SCL): btn de latest entry
   IF #btn_latest THEN
       IF #index_write > 1 THEN
           #index := #index_write - 1;
       ELSE
           #index := 100;
       END_IF;
   END_IF;

   #DisplayEntry := #logArray[#index];
END_REGION
END_FUNCTION_BLOCK

// folder: PID-uri

ORGANIZATION_BLOCK "PID_Sistem_1"   // OB30, LAD, CyclicInterrupt
{ S7_Optimized_Access := 'TRUE' }
VERSION : 0.1
   VAR_INPUT
      Initial_Call : Bool;   // Initial call of this OB
      Event_Count : Int;   // Events discarded
   END_VAR
   VAR_TEMP   // added for the SCL form of the ladder/FBD networks
      _w1 : Bool;
   END_VAR
BEGIN

REGION Network 1: block ul de PID
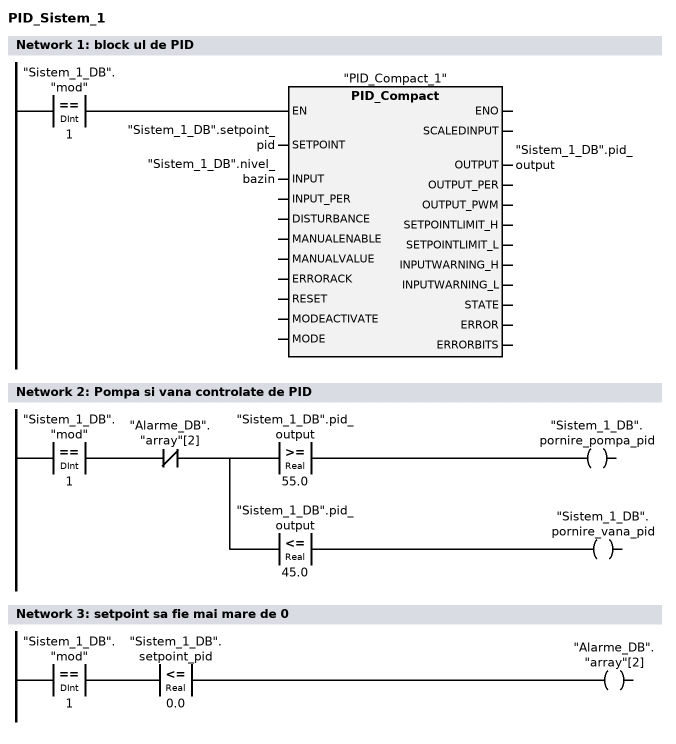
   IF "Sistem_1_DB"."mod" = 1 THEN
       "PID_Compact_1"(Setpoint := "Sistem_1_DB".setpoint_pid,   // PID_Compact
                       Input := "Sistem_1_DB".nivel_bazin,
                       Output => "Sistem_1_DB".pid_output);
   END_IF;
END_REGION

REGION Network 2: Pompa si vana controlate de PID
   RUNG wire#powerrail
      { S7_Templates := "SrcType := DInt" } EQ_Contact(in1 := "Sistem_1_DB"."mod", in2 := 1)
      I_Contact( "Alarme_DB"."array"[2] )
      wire#w1
      { S7_Templates := "SrcType := Real" } GE_Contact(in1 := "Sistem_1_DB".pid_output, in2 := 55.0)
      Coil( "Sistem_1_DB".pornire_pompa_pid )
   END_RUNG
   RUNG wire#w1
      { S7_Templates := "SrcType := Real" } LE_Contact(in1 := "Sistem_1_DB".pid_output, in2 := 45.0)
      Coil( "Sistem_1_DB".pornire_vana_pid )
   END_RUNG
   // the same network as SCL:
   #_w1 := ("Sistem_1_DB"."mod" = 1) AND NOT "Alarme_DB"."array"[2];
   "Sistem_1_DB".pornire_pompa_pid := #_w1 AND ("Sistem_1_DB".pid_output >= 55.0);
   "Sistem_1_DB".pornire_vana_pid := #_w1 AND ("Sistem_1_DB".pid_output <= 45.0);
END_REGION

REGION Network 3: setpoint sa fie mai mare de 0
   RUNG wire#powerrail
      { S7_Templates := "SrcType := DInt" } EQ_Contact(in1 := "Sistem_1_DB"."mod", in2 := 1)
      { S7_Templates := "SrcType := Real" } LE_Contact(in1 := "Sistem_1_DB".setpoint_pid, in2 := 0.0)
      Coil( "Alarme_DB"."array"[2] )
   END_RUNG
   // the same network as SCL:
   "Alarme_DB"."array"[2] := ("Sistem_1_DB"."mod" = 1) AND ("Sistem_1_DB".setpoint_pid <= 0.0);
END_REGION
END_ORGANIZATION_BLOCK

ORGANIZATION_BLOCK "PID_Sistem_2"   // OB31, LAD, CyclicInterrupt
{ S7_Optimized_Access := 'TRUE' }
VERSION : 0.1
   VAR_INPUT
      Initial_Call : Bool;   // Initial call of this OB
      Event_Count : Int;   // Events discarded
   END_VAR
   VAR_TEMP   // added for the SCL form of the ladder/FBD networks
      _w1 : Bool;
   END_VAR
BEGIN

REGION Network 1
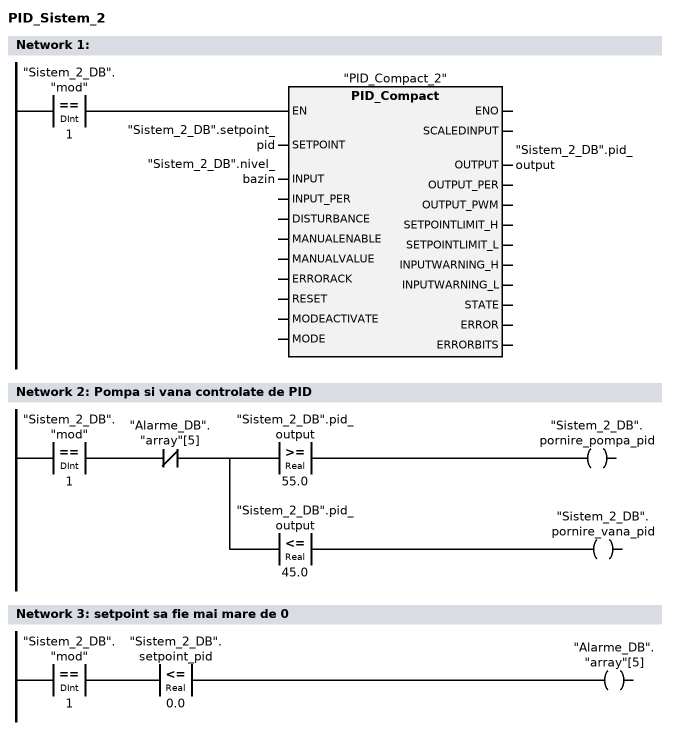
   IF "Sistem_2_DB"."mod" = 1 THEN
       "PID_Compact_2"(Setpoint := "Sistem_2_DB".setpoint_pid,   // PID_Compact
                       Input := "Sistem_2_DB".nivel_bazin,
                       Output => "Sistem_2_DB".pid_output);
   END_IF;
END_REGION

REGION Network 2: Pompa si vana controlate de PID
   RUNG wire#powerrail
      { S7_Templates := "SrcType := DInt" } EQ_Contact(in1 := "Sistem_2_DB"."mod", in2 := 1)
      I_Contact( "Alarme_DB"."array"[5] )
      wire#w1
      { S7_Templates := "SrcType := Real" } GE_Contact(in1 := "Sistem_2_DB".pid_output, in2 := 55.0)
      Coil( "Sistem_2_DB".pornire_pompa_pid )
   END_RUNG
   RUNG wire#w1
      { S7_Templates := "SrcType := Real" } LE_Contact(in1 := "Sistem_2_DB".pid_output, in2 := 45.0)
      Coil( "Sistem_2_DB".pornire_vana_pid )
   END_RUNG
   // the same network as SCL:
   #_w1 := ("Sistem_2_DB"."mod" = 1) AND NOT "Alarme_DB"."array"[5];
   "Sistem_2_DB".pornire_pompa_pid := #_w1 AND ("Sistem_2_DB".pid_output >= 55.0);
   "Sistem_2_DB".pornire_vana_pid := #_w1 AND ("Sistem_2_DB".pid_output <= 45.0);
END_REGION

REGION Network 3: setpoint sa fie mai mare de 0
   RUNG wire#powerrail
      { S7_Templates := "SrcType := DInt" } EQ_Contact(in1 := "Sistem_2_DB"."mod", in2 := 1)
      { S7_Templates := "SrcType := Real" } LE_Contact(in1 := "Sistem_2_DB".setpoint_pid, in2 := 0.0)
      Coil( "Alarme_DB"."array"[5] )
   END_RUNG
   // the same network as SCL:
   "Alarme_DB"."array"[5] := ("Sistem_2_DB"."mod" = 1) AND ("Sistem_2_DB".setpoint_pid <= 0.0);
END_REGION
END_ORGANIZATION_BLOCK

ORGANIZATION_BLOCK "PID_Sistem_3"   // OB32, LAD, CyclicInterrupt
{ S7_Optimized_Access := 'TRUE' }
VERSION : 0.1
   VAR_INPUT
      Initial_Call : Bool;   // Initial call of this OB
      Event_Count : Int;   // Events discarded
   END_VAR
   VAR_TEMP   // added for the SCL form of the ladder/FBD networks
      _w1 : Bool;
   END_VAR
BEGIN

REGION Network 1
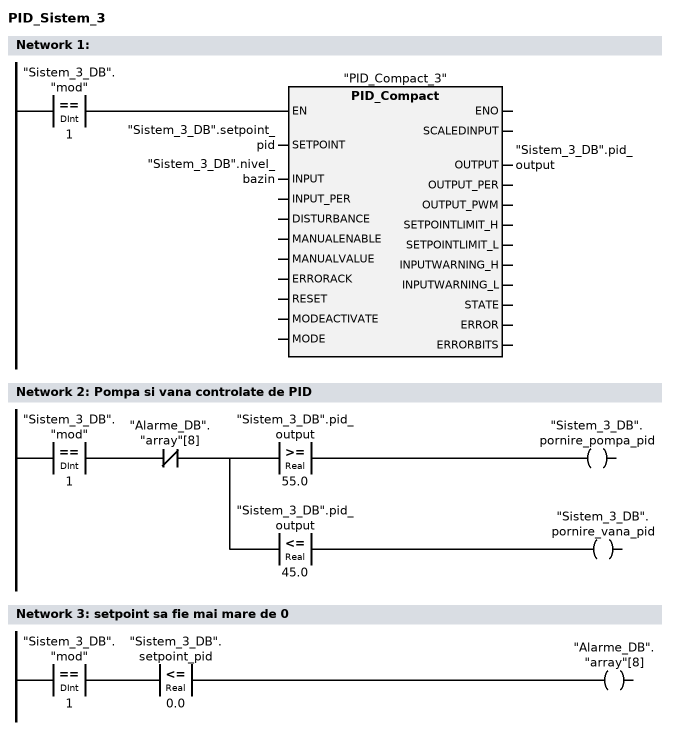
   IF "Sistem_3_DB"."mod" = 1 THEN
       "PID_Compact_3"(Setpoint := "Sistem_3_DB".setpoint_pid,   // PID_Compact
                       Input := "Sistem_3_DB".nivel_bazin,
                       Output => "Sistem_3_DB".pid_output);
   END_IF;
END_REGION

REGION Network 2: Pompa si vana controlate de PID
   RUNG wire#powerrail
      { S7_Templates := "SrcType := DInt" } EQ_Contact(in1 := "Sistem_3_DB"."mod", in2 := 1)
      I_Contact( "Alarme_DB"."array"[8] )
      wire#w1
      { S7_Templates := "SrcType := Real" } GE_Contact(in1 := "Sistem_3_DB".pid_output, in2 := 55.0)
      Coil( "Sistem_3_DB".pornire_pompa_pid )
   END_RUNG
   RUNG wire#w1
      { S7_Templates := "SrcType := Real" } LE_Contact(in1 := "Sistem_3_DB".pid_output, in2 := 45.0)
      Coil( "Sistem_3_DB".pornire_vana_pid )
   END_RUNG
   // the same network as SCL:
   #_w1 := ("Sistem_3_DB"."mod" = 1) AND NOT "Alarme_DB"."array"[8];
   "Sistem_3_DB".pornire_pompa_pid := #_w1 AND ("Sistem_3_DB".pid_output >= 55.0);
   "Sistem_3_DB".pornire_vana_pid := #_w1 AND ("Sistem_3_DB".pid_output <= 45.0);
END_REGION

REGION Network 3: setpoint sa fie mai mare de 0
   RUNG wire#powerrail
      { S7_Templates := "SrcType := DInt" } EQ_Contact(in1 := "Sistem_3_DB"."mod", in2 := 1)
      { S7_Templates := "SrcType := Real" } LE_Contact(in1 := "Sistem_3_DB".setpoint_pid, in2 := 0.0)
      Coil( "Alarme_DB"."array"[8] )
   END_RUNG
   // the same network as SCL:
   "Alarme_DB"."array"[8] := ("Sistem_3_DB"."mod" = 1) AND ("Sistem_3_DB".setpoint_pid <= 0.0);
END_REGION
END_ORGANIZATION_BLOCK

ORGANIZATION_BLOCK "PID_Sistem_4"   // OB33, LAD, CyclicInterrupt
{ S7_Optimized_Access := 'TRUE' }
VERSION : 0.1
   VAR_INPUT
      Initial_Call : Bool;   // Initial call of this OB
      Event_Count : Int;   // Events discarded
   END_VAR
   VAR_TEMP   // added for the SCL form of the ladder/FBD networks
      _w1 : Bool;
   END_VAR
BEGIN

REGION Network 1
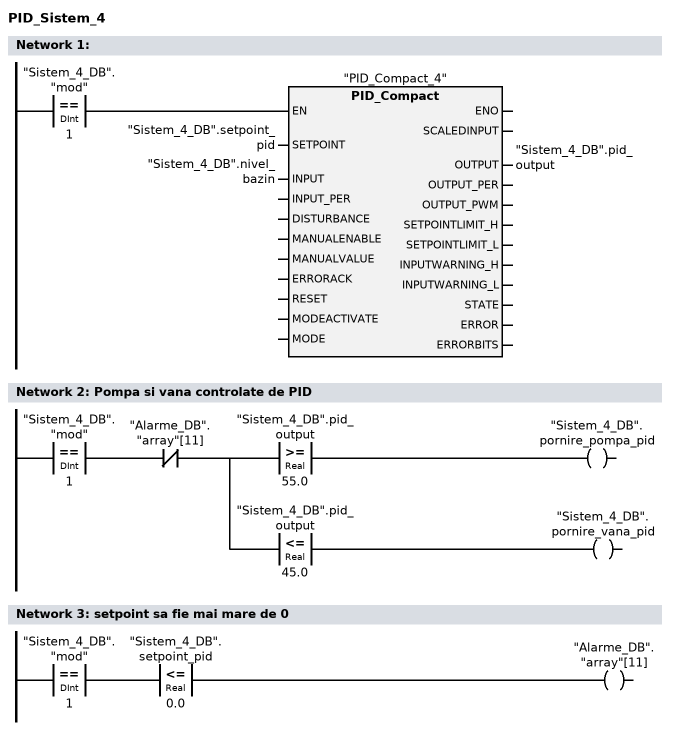
   IF "Sistem_4_DB"."mod" = 1 THEN
       "PID_Compact_4"(Setpoint := "Sistem_4_DB".setpoint_pid,   // PID_Compact
                       Input := "Sistem_4_DB".nivel_bazin,
                       Output => "Sistem_4_DB".pid_output);
   END_IF;
END_REGION

REGION Network 2: Pompa si vana controlate de PID
   RUNG wire#powerrail
      { S7_Templates := "SrcType := DInt" } EQ_Contact(in1 := "Sistem_4_DB"."mod", in2 := 1)
      I_Contact( "Alarme_DB"."array"[11] )
      wire#w1
      { S7_Templates := "SrcType := Real" } GE_Contact(in1 := "Sistem_4_DB".pid_output, in2 := 55.0)
      Coil( "Sistem_4_DB".pornire_pompa_pid )
   END_RUNG
   RUNG wire#w1
      { S7_Templates := "SrcType := Real" } LE_Contact(in1 := "Sistem_4_DB".pid_output, in2 := 45.0)
      Coil( "Sistem_4_DB".pornire_vana_pid )
   END_RUNG
   // the same network as SCL:
   #_w1 := ("Sistem_4_DB"."mod" = 1) AND NOT "Alarme_DB"."array"[11];
   "Sistem_4_DB".pornire_pompa_pid := #_w1 AND ("Sistem_4_DB".pid_output >= 55.0);
   "Sistem_4_DB".pornire_vana_pid := #_w1 AND ("Sistem_4_DB".pid_output <= 45.0);
END_REGION

REGION Network 3: setpoint sa fie mai mare de 0
   RUNG wire#powerrail
      { S7_Templates := "SrcType := DInt" } EQ_Contact(in1 := "Sistem_4_DB"."mod", in2 := 1)
      { S7_Templates := "SrcType := Real" } LE_Contact(in1 := "Sistem_4_DB".setpoint_pid, in2 := 0.0)
      Coil( "Alarme_DB"."array"[11] )
   END_RUNG
   // the same network as SCL:
   "Alarme_DB"."array"[11] := ("Sistem_4_DB"."mod" = 1) AND ("Sistem_4_DB".setpoint_pid <= 0.0);
END_REGION
END_ORGANIZATION_BLOCK

(* ===== HMI "HMI_RT_1" =====
system functions are stored by id; their names below are inferred from use
connection "HMI_Connection_1": ETHERNET, SMART_S7_1500_OMS

HMI tags "Default tag table"
   "Alarme_DB_gather" : Word = PLC Alarme_DB.gather, 1 s
   "Avarii_DB_esd_1" : Bool = PLC Avarii_DB.esd_1, 1 s
   "Sistem_1_status_pornit(HMI)" : Bool = PLC Sistem_1.status_pornit(HMI), 1 s
   "indicator_pornit_1" : Bool = PLC Sistem_1_DB.indicator_pornit AT %M10.2, 1 s
   "Avarii_DB_btn_esd_1" : Bool = PLC Avarii_DB.btn_esd_1, 1 s
   "Avarii_DB_reset_esd_1" : Bool = PLC Avarii_DB.reset_esd_1, 1 s
   "Avarii_DB_btn_avarie_sistem_1" : Bool = PLC Avarii_DB.btn_avarie_sistem_1, 1 s
   "Avarii_DB_reset_avarie_sistem_1" : Bool = PLC Avarii_DB.reset_avarie_sistem_1, 1 s
   "btn_start_1" : Bool = PLC Sistem_1_DB.btn_start AT %M100.0, 1 s
   "btn_stop_1" : Bool = PLC Sistem_1_DB.btn_stop AT %M100.1, 1 s
   "nivel_bazin_1" : Real = PLC Sistem_1_DB.nivel_bazin AT %MD0, 1 s
   "Sistem_1_mod" : DInt = PLC Sistem_1.mod, 1 s
   "mod_1" : DInt = PLC Sistem_1_DB.mod AT %MD1, 1 s
   "Sistem_1_DB_setpoint_pid" : Real = PLC Sistem_1_DB.setpoint_pid, 1 s
   "Sistem_1_DB_permisiune_start" : Bool = PLC Sistem_1_DB.permisiune_start, 1 s
   "Sistem_1_DB_plecare_pompa" : Bool = PLC Sistem_1_DB.plecare_pompa, 1 s
   "Sistem_1_DB_comanda_pornire_pompa" : Bool = PLC Sistem_1_DB.comanda_pornire_pompa, 1 s
   "Sistem_1_DB_comanda_pornire_vana" : Bool = PLC Sistem_1_DB.comanda_pornire_vana, 1 s
   "Avarii_DB_avarie_sistem_1" : Bool = PLC Avarii_DB.avarie_sistem_1, 1 s
   "Avarii_DB_esd_2" : Bool = PLC Avarii_DB.esd_2, 1 s
   "Avarii_DB_avarie_sistem_2" : Bool = PLC Avarii_DB.avarie_sistem_2, 1 s
   "Sistem_2_DB_permisiune_start" : Bool = PLC Sistem_2_DB.permisiune_start, 1 s
   "Avarii_DB_avarie_sistem_3" : Bool = PLC Avarii_DB.avarie_sistem_3, 1 s
   "Avarii_DB_avarie_sistem_4" : Bool = PLC Avarii_DB.avarie_sistem_4, 1 s
   "Avarii_DB_btn_esd_2" : Bool = PLC Avarii_DB.btn_esd_2, 1 s
   "Avarii_DB_reset_esd_2" : Bool = PLC Avarii_DB.reset_esd_2, 1 s
   "Avarii_DB_btn_avarie_sistem_2" : Bool = PLC Avarii_DB.btn_avarie_sistem_2, 1 s
   "Avarii_DB_reset_avarie_sistem_2" : Bool = PLC Avarii_DB.reset_avarie_sistem_2, 1 s
   "Sistem_2_DB_btn_start" : Bool = PLC Sistem_2_DB.btn_start, 1 s
   "Sistem_2_DB_btn_stop" : Bool = PLC Sistem_2_DB.btn_stop, 1 s
   "Sistem_2_DB_indicator_pornit" : Bool = PLC Sistem_2_DB.indicator_pornit, 1 s
   "Sistem_2_DB_mod" : DInt = PLC Sistem_2_DB.mod, 1 s
   "Sistem_2_DB_setpoint_pid" : Real = PLC Sistem_2_DB.setpoint_pid, 1 s
   "Sistem_2_DB_comanda_pornire_pompa" : Bool = PLC Sistem_2_DB.comanda_pornire_pompa, 1 s
   "Sistem_2_DB_comanda_pornire_vana" : Bool = PLC Sistem_2_DB.comanda_pornire_vana, 1 s
   "Sistem_2_DB_nivel_bazin" : Real = PLC Sistem_2_DB.nivel_bazin, 1 s
   "Avarii_DB_esd_3" : Bool = PLC Avarii_DB.esd_3, 1 s
   "Avarii_DB_btn_esd_3" : Bool = PLC Avarii_DB.btn_esd_3, 1 s
   "Avarii_DB_reset_esd_3" : Bool = PLC Avarii_DB.reset_esd_3, 1 s
   "Avarii_DB_btn_avarie_sistem_3" : Bool = PLC Avarii_DB.btn_avarie_sistem_3, 1 s
   "Avarii_DB_reset_avarie_sistem_3" : Bool = PLC Avarii_DB.reset_avarie_sistem_3, 1 s
   "Sistem_3_DB_btn_start" : Bool = PLC Sistem_3_DB.btn_start, 1 s
   "Sistem_3_DB_btn_stop" : Bool = PLC Sistem_3_DB.btn_stop, 1 s
   "Sistem_3_DB_indicator_pornit" : Bool = PLC Sistem_3_DB.indicator_pornit, 1 s
   "Sistem_3_DB_mod" : DInt = PLC Sistem_3_DB.mod, 1 s
   "Sistem_3_DB_nivel_bazin" : Real = PLC Sistem_3_DB.nivel_bazin, 1 s
   "Sistem_3_DB_setpoint_pid" : Real = PLC Sistem_3_DB.setpoint_pid, 1 s
   "Sistem_3_DB_comanda_pornire_pompa" : Bool = PLC Sistem_3_DB.comanda_pornire_pompa, 1 s
   "Sistem_3_DB_comanda_pornire_vana" : Bool = PLC Sistem_3_DB.comanda_pornire_vana, 1 s
   "Avarii_DB_esd_4" : Bool = PLC Avarii_DB.esd_4, 1 s
   "Avarii_DB_btn_esd_4" : Bool = PLC Avarii_DB.btn_esd_4, 1 s
   "Avarii_DB_reset_esd_4" : Bool = PLC Avarii_DB.reset_esd_4, 1 s
   "Avarii_DB_reset_avarie_sistem_4" : Bool = PLC Avarii_DB.reset_avarie_sistem_4, 1 s
   "Avarii_DB_btn_avarie_sistem_4" : Bool = PLC Avarii_DB.btn_avarie_sistem_4, 1 s
   "Sistem_4_DB_btn_start" : Bool = PLC Sistem_4_DB.btn_start, 1 s
   "Sistem_4_DB_btn_stop" : Bool = PLC Sistem_4_DB.btn_stop, 1 s
   "Sistem_4_DB_indicator_pornit" : Bool = PLC Sistem_4_DB.indicator_pornit, 1 s
   "Sistem_4_DB_nivel_bazin" : Real = PLC Sistem_4_DB.nivel_bazin, 1 s
   "Sistem_4_DB_mod" : DInt = PLC Sistem_4_DB.mod, 1 s
   "Sistem_4_DB_setpoint_pid" : Real = PLC Sistem_4_DB.setpoint_pid, 1 s
   "Sistem_4_DB_comanda_pornire_pompa" : Bool = PLC Sistem_4_DB.comanda_pornire_pompa, 1 s
   "Sistem_4_DB_comanda_pornire_vana" : Bool = PLC Sistem_4_DB.comanda_pornire_vana, 1 s
   "Sistem_3_DB_permisiune_start" : Bool = PLC Sistem_3_DB.permisiune_start, 1 s
   "Sistem_4_DB_permisiune_start" : Bool = PLC Sistem_4_DB.permisiune_start, 1 s
   "Logs1_DB_index" : Int = PLC Logs1_DB.index, 1 s
   "Logs1_DB_target_index" : Int = PLC Logs1_DB.target_index, 1 s
   "Logs1_DB_Display_Entry_Timestamp_SECOND" : USInt = PLC Logs1_DB.Display_Entry.Timestamp.SECOND, 1 s
   "Logs1_DB_Display_Entry_Timestamp_MINUTE" : USInt = PLC Logs1_DB.Display_Entry.Timestamp.MINUTE, 1 s
   "Logs1_DB_Display_Entry_Timestamp_HOUR" : USInt = PLC Logs1_DB.Display_Entry.Timestamp.HOUR, 1 s
   "Logs1_DB_Display_Entry_Timestamp_DAY" : USInt = PLC Logs1_DB.Display_Entry.Timestamp.DAY, 1 s
   "Logs1_DB_Display_Entry_Timestamp" : DTL = PLC Logs1_DB.Display_Entry.Timestamp, 1 s
   "Logs1_DB_Display_Entry_Level" : Real = PLC Logs1_DB.Display_Entry.Level, 1 s
   "Logs1_DB_Display_Entry_Mode" : DInt = PLC Logs1_DB.Display_Entry.Mode, 1 s
   "Logs1_DB_Display_Entry_ESD_Active" : Bool = PLC Logs1_DB.Display_Entry.ESD_Active, 1 s
   "Logs1_DB_Display_Entry_Fault_Active" : Bool = PLC Logs1_DB.Display_Entry.Fault_Active, 1 s
   "Logs1_DB_btn_jump" : Bool = PLC Logs1_DB.btn_jump, 1 s
   "Logs1_DB_btn_prev" : Bool = PLC Logs1_DB.btn_prev, 1 s
   "Logs1_DB_btn_next" : Bool = PLC Logs1_DB.btn_next, 1 s
   "Logs1_DB_btn_latest" : Bool = PLC Logs1_DB.btn_latest, 1 s
   "Logs2_DB_index" : Int = PLC Logs2_DB.index, 1 s
   "Logs2_DB_Display_Entry_Timestamp" : DTL = PLC Logs2_DB.Display_Entry.Timestamp, 1 s
   "Logs2_DB_Display_Entry_Level" : Real = PLC Logs2_DB.Display_Entry.Level, 1 s
   "Logs2_DB_Display_Entry_Mode" : DInt = PLC Logs2_DB.Display_Entry.Mode, 1 s
   "Logs2_DB_Display_Entry_ESD_Active" : Bool = PLC Logs2_DB.Display_Entry.ESD_Active, 1 s
   "Logs2_DB_Display_Entry_Fault_Active" : Bool = PLC Logs2_DB.Display_Entry.Fault_Active, 1 s
   "Logs2_DB_target_index" : Int = PLC Logs2_DB.target_index, 1 s
   "Logs2_DB_btn_jump" : Bool = PLC Logs2_DB.btn_jump, 1 s
   "Logs2_DB_btn_latest" : Bool = PLC Logs2_DB.btn_latest, 1 s
   "Logs2_DB_btn_prev" : Bool = PLC Logs2_DB.btn_prev, 1 s
   "Logs2_DB_btn_next" : Bool = PLC Logs2_DB.btn_next, 1 s
   "Logs3_DB_index" : Int = PLC Logs3_DB.index, 1 s
   "Logs3_DB_Display_Entry_Timestamp" : DTL = PLC Logs3_DB.Display_Entry.Timestamp, 1 s
   "Logs3_DB_Display_Entry_Level" : Real = PLC Logs3_DB.Display_Entry.Level, 1 s
   "Logs3_DB_Display_Entry_Mode" : DInt = PLC Logs3_DB.Display_Entry.Mode, 1 s
   "Logs3_DB_Display_Entry_ESD_Active" : Bool = PLC Logs3_DB.Display_Entry.ESD_Active, 1 s
   "Logs3_DB_Display_Entry_Fault_Active" : Bool = PLC Logs3_DB.Display_Entry.Fault_Active, 1 s
   "Logs3_DB_target_index" : Int = PLC Logs3_DB.target_index, 1 s
   "Logs3_DB_btn_jump" : Bool = PLC Logs3_DB.btn_jump, 1 s
   "Logs3_DB_btn_latest" : Bool = PLC Logs3_DB.btn_latest, 1 s
   "Logs3_DB_btn_prev" : Bool = PLC Logs3_DB.btn_prev, 1 s
   "Logs3_DB_btn_next" : Bool = PLC Logs3_DB.btn_next, 1 s
   "Logs4_DB_index" : Int = PLC Logs4_DB.index, 1 s
   "Logs4_DB_Display_Entry_Timestamp" : DTL = PLC Logs4_DB.Display_Entry.Timestamp, 1 s
   "Logs4_DB_Display_Entry_Level" : Real = PLC Logs4_DB.Display_Entry.Level, 1 s
   "Logs4_DB_Display_Entry_Mode" : DInt = PLC Logs4_DB.Display_Entry.Mode, 1 s
   "Logs4_DB_Display_Entry_ESD_Active" : Bool = PLC Logs4_DB.Display_Entry.ESD_Active, 1 s
   "Logs4_DB_Display_Entry_Fault_Active" : Bool = PLC Logs4_DB.Display_Entry.Fault_Active, 1 s
   "Logs4_DB_target_index" : Int = PLC Logs4_DB.target_index, 1 s
   "Logs4_DB_btn_jump" : Bool = PLC Logs4_DB.btn_jump, 1 s
   "Logs4_DB_btn_latest" : Bool = PLC Logs4_DB.btn_latest, 1 s
   "Logs4_DB_btn_prev" : Bool = PLC Logs4_DB.btn_prev, 1 s
   "Logs4_DB_btn_next" : Bool = PLC Logs4_DB.btn_next, 1 s

discrete alarms
   1: 'ESD sistem 1', class Errors, trigger "Alarme_DB_gather" bit 0
   2: 'Avarie sistem 1', class Errors, trigger "Alarme_DB_gather" bit 1
   3: 'Setpoint-ul la PID nu este setat la sistemul 1', class Errors, trigger "Alarme_DB_gather" bit 2
   4: 'ESD sistem 2', class Errors, trigger "Alarme_DB_gather" bit 3
   5: 'Avarie sistem 2', class Errors, trigger "Alarme_DB_gather" bit 4
   6: 'Setpoint-ul la PID nu este setat la sistemul 2', class Errors, trigger "Alarme_DB_gather" bit 5
   7: 'ESD sistem 3', class Errors, trigger "Alarme_DB_gather" bit 6
   8: 'Avarie sistem 3', class Errors, trigger "Alarme_DB_gather" bit 7
   9: 'Setpoint-ul la PID nu este setat la sistemul 3', class Errors, trigger "Alarme_DB_gather" bit 8
   10: 'ESD sistem 4', class Errors, trigger "Alarme_DB_gather" bit 9
   11: 'Avarie sistem 4', class Errors, trigger "Alarme_DB_gather" bit 10
   12: 'Setpoint-ul la PID nu este setat la sistemul 4', class Errors, trigger "Alarme_DB_gather" bit 11

text list "Moduri": 0 'Manual'; 1 'Automat'

screen "Pompa1" 800x480, template "Template_1"
   TextField "Text field_1" at 23,455 size 60x20; Text 'Pompa 1'
   TextField "Text field_2" at 121,455 size 60x20; Text 'Pompa 2'
   TextField "Text field_3" at 221,455 size 60x20; Text 'Pompa 3'
   TextField "Text field_4" at 321,455 size 60x20; Text 'Pompa 4'
   TextField "Text field_5" at 429,455 size 43x20; Text 'Logs1'
   TrendView "Trend view_1" at 0,217 size 800x225
   Bar "Bar_1" at 582,56 size 165x149; MinimumValue 0; MaximumValue 100
      ProcessValue <- "nivel_bazin_1"
   IOField "I/O field_1" at 618,24 size 96x32; FormatPattern 999.99; Unit L
      ProcessValue <- "nivel_bazin_1"
   TextField "Text field_6" at 357,3 size 88x27; Text 'Pompa 1'
   TextField "Text field_7" at 646,4 size 39x20; Text 'Bazin'
   Button "Button_1" at 26,115 size 55x32; TextOff 'ESD'
      on Click: SetBit("Avarii_DB_btn_esd_1")
   Button "Button_2" at 26,147 size 55x32; TextOff 'Reset'
      on Click: SetBit("Avarii_DB_reset_esd_1")
   Circle "Circle_1" at 30,55 size 48x48
      Appearance <- "Avarii_DB_esd_1"
   SymbolicIOField "Symbolic I/O field_1" at 351,73 size 101x32; TextOff '0'; TextOn '1'; TextList "Moduri"
      ProcessValue <- "mod_1"
   Button "Button_3" at 105,115 size 55x32; TextOff 'Avarie'
      on Press: SetBit("Avarii_DB_btn_avarie_sistem_1")
   Button "Button_4" at 105,147 size 55x32; TextOff 'Reset'
      on Click: SetBit("Avarii_DB_reset_avarie_sistem_1")
   Circle "Circle_2" at 109,55 size 48x48
      Appearance <- "Avarii_DB_avarie_sistem_1"
   IOField "I/O field_2" at 351,135 size 101x32; FormatPattern 999.99; Unit L
      Visibility <- "mod_1"
      ProcessValue <- "Sistem_1_DB_setpoint_pid"
   TextField "Text field_8" at 383,52 size 32x20; Text 'Mod'
   TextField "Text field_9" at 358,115 size 86x20; Text 'Setpoint PID'
      Visibility <- "mod_1"
   Button "Button_5" at 480,75 size 27x28; TextOff 'On'
      Visibility <- "mod_1"
      on Press: SetTag("Sistem_1_DB_comanda_pornire_pompa", 1)
      Appearance <- "Sistem_1_DB_comanda_pornire_pompa"
   Button "Button_6" at 511,75 size 27x28; TextOff 'Off'
      Visibility <- "mod_1"
      on Press: SetTag("Sistem_1_DB_comanda_pornire_pompa", 0)
      Appearance <- "Sistem_1_DB_comanda_pornire_pompa"
   TextField "Text field_10" at 485,54 size 48x20; Text 'Pompa'
      Visibility <- "mod_1"
   Button "Button_7" at 480,126 size 27x28; TextOff 'On'
      Visibility <- "mod_1"
      on Press: SetTag("Sistem_1_DB_comanda_pornire_vana", 1)
      Appearance <- "Sistem_1_DB_comanda_pornire_vana"
   Button "Button_8" at 511,126 size 27x28; TextOff 'Off'
      Visibility <- "mod_1"
      on Press: SetTag("Sistem_1_DB_comanda_pornire_vana", 0)
      Appearance <- "Sistem_1_DB_comanda_pornire_vana"
   TextField "Text field_11" at 489,105 size 38x20; Text 'Vana'
      Visibility <- "mod_1"
   Circle "Circle_3" at 189,55 size 48x48
      Appearance <- "Sistem_1_DB_permisiune_start"
   TextField "Text field_13" at 275,59 size 44x20; Text 'Pornit'
   Button "Button_9" at 189,115 size 46x32; TextOff 'Start'
      on Click: SetBit("btn_start_1")
   Button "Button_10" at 189,147 size 46x32; TextOff 'Stop'
      on Click: SetBit("btn_stop_1")
   Circle "Circle_4" at 267,88 size 61x61
      Appearance <- "indicator_pornit_1"
   TextField "Text field_12" at 528,454 size 43x20; Text 'Logs2'
   TextField "Text field_14" at 627,453 size 43x20; Text 'Logs3'
   TextField "Text field_15" at 726,452 size 43x20; Text 'Logs4'

screen "Pompa2" 800x480
   TextField "Text field_1" at 23,455 size 60x20; Text 'Pompa 1'
   TextField "Text field_2" at 121,455 size 60x20; Text 'Pompa 2'
   TextField "Text field_3" at 221,455 size 60x20; Text 'Pompa 3'
   TextField "Text field_4" at 321,455 size 60x20; Text 'Pompa 4'
   TrendView "Trend view_1" at 0,217 size 800x225
   Bar "Bar_1" at 582,56 size 165x149; MinimumValue 0; MaximumValue 100
      ProcessValue <- "Sistem_2_DB_nivel_bazin"
   IOField "I/O field_1" at 618,24 size 96x32; FormatPattern 999.99; Unit L
      ProcessValue <- "Sistem_2_DB_nivel_bazin"
   TextField "Text field_11" at 357,3 size 88x27; Text 'Pompa 2'
   TextField "Text field_12" at 646,4 size 39x20; Text 'Bazin'
   Button "Button_1" at 26,115 size 55x32; TextOff 'ESD'
      on Click: SetBit("Avarii_DB_btn_esd_2")
   Button "Button_2" at 26,147 size 55x32; TextOff 'Reset'
      on Click: SetBit("Avarii_DB_reset_esd_2")
   Circle "Circle_1" at 30,55 size 48x48
      Appearance <- "Avarii_DB_esd_2"
   SymbolicIOField "Symbolic I/O field_1" at 351,73 size 101x32; TextOn '1'; TextOff '0'; TextList "Moduri"
      ProcessValue <- "Sistem_2_DB_mod"
   Button "Button_3" at 105,115 size 55x32; TextOff 'Avarie'
      on Press: SetBit("Avarii_DB_btn_avarie_sistem_2")
   Button "Button_4" at 105,147 size 55x32; TextOff 'Reset'
      on Click: SetBit("Avarii_DB_reset_avarie_sistem_2")
   Circle "Circle_2" at 109,55 size 48x48
      Appearance <- "Avarii_DB_avarie_sistem_2"
   IOField "I/O field_2" at 351,135 size 101x32; FormatPattern 999.99; Unit L
      ProcessValue <- "Sistem_2_DB_setpoint_pid"
      Visibility <- "Sistem_2_DB_mod"
   TextField "Text field_13" at 383,52 size 32x20; Text 'Mod'
   TextField "Text field_14" at 358,115 size 86x20; Text 'Setpoint PID'
      Visibility <- "Sistem_2_DB_mod"
   Button "Button_5" at 480,75 size 27x28; TextOff 'On'
      on Press: SetTag("Sistem_2_DB_comanda_pornire_pompa", 1)
      Visibility <- "Sistem_2_DB_mod"
      Appearance <- "Sistem_2_DB_comanda_pornire_pompa"
   Button "Button_6" at 511,75 size 27x28; TextOff 'Off'
      on Press: SetTag("Sistem_2_DB_comanda_pornire_pompa", 0)
      Visibility <- "Sistem_2_DB_mod"
      Appearance <- "Sistem_2_DB_comanda_pornire_pompa"
   TextField "Text field_15" at 485,54 size 48x20; Text 'Pompa'
      Visibility <- "Sistem_2_DB_mod"
   Button "Button_7" at 480,126 size 27x28; TextOff 'On'
      on Press: SetTag("Sistem_2_DB_comanda_pornire_vana", 1)
      Visibility <- "Sistem_2_DB_mod"
      Appearance <- "Sistem_2_DB_comanda_pornire_vana"
   Button "Button_8" at 511,126 size 27x28; TextOff 'Off'
      on Press: SetTag("Sistem_2_DB_comanda_pornire_vana", 0)
      Visibility <- "Sistem_2_DB_mod"
      Appearance <- "Sistem_2_DB_comanda_pornire_vana"
   TextField "Text field_16" at 489,105 size 38x20; Text 'Vana'
      Visibility <- "Sistem_2_DB_mod"
   Circle "Circle_3" at 189,55 size 48x48
      Appearance <- "Sistem_2_DB_permisiune_start"
   TextField "Text field_17" at 275,59 size 44x20; Text 'Pornit'
   Button "Button_9" at 189,115 size 46x32; TextOff 'Start'
      on Click: SetBit("Sistem_2_DB_btn_start")
   Button "Button_10" at 189,147 size 46x32; TextOff 'Stop'
      on Click: SetBit("Sistem_2_DB_btn_stop")
   Circle "Circle_4" at 267,88 size 61x61
      Appearance <- "Sistem_2_DB_indicator_pornit"
   TextField "Text field_5" at 429,455 size 43x20; Text 'Logs1'
   TextField "Text field_6" at 528,454 size 43x20; Text 'Logs2'
   TextField "Text field_7" at 627,453 size 43x20; Text 'Logs3'
   TextField "Text field_8" at 726,452 size 43x20; Text 'Logs4'

screen "Pompa3" 800x480
   TextField "Text field_1" at 23,455 size 60x20; Text 'Pompa 1'
   TextField "Text field_2" at 121,455 size 60x20; Text 'Pompa 2'
   TextField "Text field_3" at 221,455 size 60x20; Text 'Pompa 3'
   TextField "Text field_4" at 321,455 size 60x20; Text 'Pompa 4'
   TrendView "Trend view_1" at 0,217 size 800x225
   Bar "Bar_1" at 582,56 size 165x149; MinimumValue 0; MaximumValue 100
      ProcessValue <- "Sistem_3_DB_nivel_bazin"
   IOField "I/O field_1" at 618,24 size 96x32; FormatPattern 999.99; Unit L
      ProcessValue <- "Sistem_3_DB_nivel_bazin"
   TextField "Text field_6" at 357,3 size 88x27; Text 'Pompa 3'
   TextField "Text field_7" at 646,4 size 39x20; Text 'Bazin'
   Button "Button_1" at 26,115 size 55x32; TextOff 'ESD'
      on Click: SetBit("Avarii_DB_btn_esd_3")
   Button "Button_2" at 26,147 size 55x32; TextOff 'Reset'
      on Click: SetBit("Avarii_DB_reset_esd_3")
   Circle "Circle_1" at 30,55 size 48x48
      Appearance <- "Avarii_DB_esd_3"
   SymbolicIOField "Symbolic I/O field_1" at 351,73 size 101x32; TextOn '1'; TextOff '0'; TextList "Moduri"
      ProcessValue <- "Sistem_3_DB_mod"
   Button "Button_3" at 105,115 size 55x32; TextOff 'Avarie'
      on Press: SetBit("Avarii_DB_btn_avarie_sistem_3")
   Button "Button_4" at 105,147 size 55x32; TextOff 'Reset'
      on Click: SetBit("Avarii_DB_reset_avarie_sistem_3")
   Circle "Circle_2" at 109,55 size 48x48
      Appearance <- "Avarii_DB_avarie_sistem_3"
   IOField "I/O field_2" at 351,135 size 101x32; FormatPattern 999.99; Unit L
      Visibility <- "Sistem_3_DB_mod"
      ProcessValue <- "Sistem_3_DB_setpoint_pid"
   TextField "Text field_8" at 383,52 size 32x20; Text 'Mod'
   TextField "Text field_9" at 358,115 size 86x20; Text 'Setpoint PID'
      Visibility <- "Sistem_3_DB_mod"
   TextField "Text field_10" at 485,54 size 48x20; Text 'Pompa'
      Visibility <- "Sistem_3_DB_mod"
   TextField "Text field_11" at 489,105 size 38x20; Text 'Vana'
      Visibility <- "Sistem_3_DB_mod"
   Circle "Circle_3" at 189,55 size 48x48
      Appearance <- "Sistem_3_DB_permisiune_start"
   TextField "Text field_13" at 275,59 size 44x20; Text 'Pornit'
   Button "Button_9" at 189,115 size 46x32; TextOff 'Start'
      on Click: SetBit("Sistem_3_DB_btn_start")
   Button "Button_10" at 189,147 size 46x32; TextOff 'Stop'
      on Click: SetBit("Sistem_3_DB_btn_stop")
   Circle "Circle_4" at 267,88 size 61x61
      Appearance <- "Sistem_3_DB_indicator_pornit"
   Button "Button_5" at 480,75 size 27x28; TextOff 'On'
      on Press: SetTag("Sistem_3_DB_comanda_pornire_pompa", 1)
      Visibility <- "Sistem_3_DB_mod"
      Appearance <- "Sistem_3_DB_comanda_pornire_pompa"
   Button "Button_6" at 511,75 size 27x28; TextOff 'Off'
      on Press: SetTag("Sistem_3_DB_comanda_pornire_pompa", 0)
      Visibility <- "Sistem_3_DB_mod"
      Appearance <- "Sistem_3_DB_comanda_pornire_pompa"
   Button "Button_7" at 480,126 size 27x28; TextOff 'On'
      on Press: SetTag("Sistem_3_DB_comanda_pornire_vana", 1)
      Visibility <- "Sistem_3_DB_mod"
      Appearance <- "Sistem_3_DB_comanda_pornire_vana"
   Button "Button_8" at 511,126 size 27x28; TextOff 'Off'
      on Press: SetTag("Sistem_3_DB_comanda_pornire_vana", 0)
      Visibility <- "Sistem_3_DB_mod"
      Appearance <- "Sistem_3_DB_comanda_pornire_vana"
   TextField "Text field_5" at 429,455 size 43x20; Text 'Logs1'
   TextField "Text field_12" at 528,454 size 43x20; Text 'Logs2'
   TextField "Text field_14" at 627,453 size 43x20; Text 'Logs3'
   TextField "Text field_15" at 726,452 size 43x20; Text 'Logs4'

screen "Pompa4" 800x480
   TextField "Text field_1" at 23,455 size 60x20; Text 'Pompa 1'
   TextField "Text field_2" at 121,455 size 60x20; Text 'Pompa 2'
   TextField "Text field_3" at 221,455 size 60x20; Text 'Pompa 3'
   TextField "Text field_4" at 321,455 size 60x20; Text 'Pompa 4'
   TrendView "Trend view_1" at 0,217 size 800x225
   Bar "Bar_1" at 582,56 size 165x149; MinimumValue 0; MaximumValue 100
      ProcessValue <- "Sistem_4_DB_nivel_bazin"
   IOField "I/O field_1" at 618,24 size 96x32; FormatPattern 999.99; Unit L
      ProcessValue <- "Sistem_4_DB_nivel_bazin"
   TextField "Text field_6" at 357,3 size 88x27; Text 'Pompa 4'
   TextField "Text field_7" at 646,4 size 39x20; Text 'Bazin'
   Button "Button_1" at 26,115 size 55x32; TextOff 'ESD'
      on Click: SetBit("Avarii_DB_btn_esd_4")
   Button "Button_2" at 26,147 size 55x32; TextOff 'Reset'
      on Click: SetBit("Avarii_DB_reset_esd_4")
   Circle "Circle_1" at 30,55 size 48x48
      Appearance <- "Avarii_DB_esd_4"
   SymbolicIOField "Symbolic I/O field_1" at 351,73 size 101x32; TextOn '1'; TextOff '0'; TextList "Moduri"
      ProcessValue <- "Sistem_4_DB_mod"
   Button "Button_3" at 105,115 size 55x32; TextOff 'Avarie'
      on Press: SetBit("Avarii_DB_btn_avarie_sistem_4")
   Button "Button_4" at 105,147 size 55x32; TextOff 'Reset'
      on Click: SetBit("Avarii_DB_reset_avarie_sistem_4")
   Circle "Circle_2" at 109,55 size 48x48
      Appearance <- "Avarii_DB_avarie_sistem_4"
   IOField "I/O field_2" at 351,135 size 101x32; FormatPattern 999.99; Unit L
      Visibility <- "Sistem_4_DB_mod"
      ProcessValue <- "Sistem_4_DB_setpoint_pid"
   TextField "Text field_8" at 383,52 size 32x20; Text 'Mod'
   TextField "Text field_9" at 358,115 size 86x20; Text 'Setpoint PID'
      Visibility <- "Sistem_4_DB_mod"
   TextField "Text field_10" at 485,54 size 48x20; Text 'Pompa'
      Visibility <- "Sistem_4_DB_mod"
   TextField "Text field_11" at 489,105 size 38x20; Text 'Vana'
      Visibility <- "Sistem_4_DB_mod"
   Circle "Circle_3" at 189,55 size 48x48
      Appearance <- "Sistem_4_DB_permisiune_start"
   TextField "Text field_13" at 275,59 size 44x20; Text 'Pornit'
   Button "Button_9" at 189,115 size 46x32; TextOff 'Start'
      on Click: SetBit("Sistem_4_DB_btn_start")
   Button "Button_10" at 189,147 size 46x32; TextOff 'Stop'
      on Click: SetBit("Sistem_4_DB_btn_stop")
   Circle "Circle_4" at 267,88 size 61x61
      Appearance <- "Sistem_4_DB_indicator_pornit"
   Button "Button_5" at 480,75 size 27x28; TextOff 'On'
      on Press: SetTag("Sistem_4_DB_comanda_pornire_pompa", 1)
      Visibility <- "Sistem_4_DB_mod"
      Appearance <- "Sistem_4_DB_comanda_pornire_pompa"
   Button "Button_6" at 511,75 size 27x28; TextOff 'Off'
      on Press: SetTag("Sistem_4_DB_comanda_pornire_pompa", 0)
      Visibility <- "Sistem_4_DB_mod"
      Appearance <- "Sistem_4_DB_comanda_pornire_pompa"
   Button "Button_7" at 480,126 size 27x28; TextOff 'On'
      on Press: SetTag("Sistem_4_DB_comanda_pornire_vana", 1)
      Visibility <- "Sistem_4_DB_mod"
      Appearance <- "Sistem_4_DB_comanda_pornire_vana"
   Button "Button_8" at 511,126 size 27x28; TextOff 'Off'
      on Press: SetTag("Sistem_4_DB_comanda_pornire_vana", 0)
      Visibility <- "Sistem_4_DB_mod"
      Appearance <- "Sistem_4_DB_comanda_pornire_vana"
   TextField "Text field_5" at 429,455 size 43x20; Text 'Logs1'
   TextField "Text field_12" at 528,454 size 43x20; Text 'Logs2'
   TextField "Text field_14" at 627,453 size 43x20; Text 'Logs3'
   TextField "Text field_15" at 726,452 size 43x20; Text 'Logs4'

screen "Logs1" 800x480
   TextField "Text field_1" at 23,455 size 60x20; Text 'Pompa 1'
   TextField "Text field_2" at 121,455 size 60x20; Text 'Pompa 2'
   TextField "Text field_3" at 221,455 size 60x20; Text 'Pompa 3'
   TextField "Text field_4" at 321,455 size 60x20; Text 'Pompa 4'
   TextField "Text field_5" at 429,455 size 43x20; Text 'Logs1'
   TextField "Text field_12" at 528,454 size 43x20; Text 'Logs2'
   TextField "Text field_14" at 627,453 size 43x20; Text 'Logs3'
   TextField "Text field_15" at 726,452 size 43x20; Text 'Logs4'
   TextField "Text field_11" at 357,3 size 68x27; Text 'Logs 1'
   TextField "Text field_6" at 552,65 size 98x20; Text 'Index Curent:'
   IOField "I/O field_1" at 647,63 size 29x25; FormatPattern 999
      ProcessValue <- "Logs1_DB_index"
   Button "Button_1" at 633,374 size 56x29; TextOff 'Inainte'
      on Press: SetBit("Logs1_DB_btn_next")
      on Release: ResetBit("Logs1_DB_btn_next")
   Button "Button_2" at 569,374 size 56x29; TextOff 'Inapoi'
      on Press: SetBit("Logs1_DB_btn_prev")
      on Release: ResetBit("Logs1_DB_btn_prev")
   TextField "Text field_7" at 127,377 size 88x20; Text 'Sari la index:'
   IOField "I/O field_2" at 220,375 size 29x25; FormatPattern 999
      ProcessValue <- "Logs1_DB_target_index"
   Button "Button_3" at 257,374 size 56x29; TextOff 'Gaseste'
      on Press: SetBit("Logs1_DB_btn_jump")
      on Release: ResetBit("Logs1_DB_btn_jump")
   TextField "Text field_8" at 177,176 size 65x29; Text 'Nivel:'
   IOField "I/O field_3" at 244,176 size 96x32; FormatPattern 999.99
      ProcessValue <- "Logs1_DB_Display_Entry_Level"
   TextField "Text field_9" at 446,179 size 58x29; Text 'Mod:'
   IOField "I/O field_4" at 510,179 size 96x32; FormatPattern 99
      ProcessValue <- "Logs1_DB_Display_Entry_Mode"
   TextField "Text field_10" at 175,120 size 130x29; Text 'Timestamp:'
   TextField "Text field_13" at 177,236 size 55x29; Text 'ESD:'
   IOField "I/O field_6" at 237,236 size 96x32; FormatPattern 1
      ProcessValue <- "Logs1_DB_Display_Entry_ESD_Active"
   TextField "Text field_16" at 446,239 size 79x29; Text 'Avarie:'
   IOField "I/O field_7" at 527,239 size 96x32; FormatPattern 1
      ProcessValue <- "Logs1_DB_Display_Entry_Fault_Active"
   IOField "I/O field_11" at 309,120 size 304x32; FormatPattern 9999999999999999999999999999999999999999
      ProcessValue <- "Logs1_DB_Display_Entry_Timestamp"
   Button "Button_4" at 463,374 size 56x29; TextOff 'Gaseste'
      on Release: ResetBit("Logs1_DB_btn_latest")
      on Press: SetBit("Logs1_DB_btn_latest")
   TextField "Text field_17" at 361,378 size 98x20; Text 'Ultima intrare:'

screen "Logs2" 800x480
   TextField "Text field_1" at 23,455 size 60x20; Text 'Pompa 1'
   TextField "Text field_2" at 121,455 size 60x20; Text 'Pompa 2'
   TextField "Text field_3" at 221,455 size 60x20; Text 'Pompa 3'
   TextField "Text field_4" at 321,455 size 60x20; Text 'Pompa 4'
   TextField "Text field_5" at 429,455 size 43x20; Text 'Logs1'
   TextField "Text field_12" at 528,454 size 43x20; Text 'Logs2'
   TextField "Text field_14" at 627,453 size 43x20; Text 'Logs3'
   TextField "Text field_15" at 726,452 size 43x20; Text 'Logs4'
   TextField "Text field_11" at 357,3 size 68x27; Text 'Logs 2'
   TextField "Text field_6" at 552,65 size 98x20; Text 'Index Curent:'
   IOField "I/O field_1" at 647,63 size 29x25; FormatPattern 999
      ProcessValue <- "Logs2_DB_index"
   Button "Button_1" at 633,374 size 56x29; TextOff 'Inainte'
      on Release: ResetBit("Logs2_DB_btn_next")
      on Press: SetBit("Logs2_DB_btn_next")
   Button "Button_2" at 569,374 size 56x29; TextOff 'Inapoi'
      on Release: ResetBit("Logs2_DB_btn_prev")
      on Press: SetBit("Logs2_DB_btn_prev")
   TextField "Text field_7" at 127,377 size 88x20; Text 'Sari la index:'
   IOField "I/O field_2" at 220,375 size 29x25; FormatPattern 999
      ProcessValue <- "Logs2_DB_target_index"
   Button "Button_3" at 257,374 size 56x29; TextOff 'Gaseste'
      on Release: ResetBit("Logs2_DB_btn_jump")
      on Press: SetBit("Logs2_DB_btn_jump")
   TextField "Text field_8" at 177,176 size 65x29; Text 'Nivel:'
   IOField "I/O field_3" at 244,176 size 96x32; FormatPattern 999.99
      ProcessValue <- "Logs2_DB_Display_Entry_Level"
   TextField "Text field_9" at 446,179 size 58x29; Text 'Mod:'
   IOField "I/O field_4" at 510,179 size 96x32; FormatPattern 99
      ProcessValue <- "Logs2_DB_Display_Entry_Mode"
   TextField "Text field_10" at 175,120 size 130x29; Text 'Timestamp:'
   TextField "Text field_13" at 177,236 size 55x29; Text 'ESD:'
   IOField "I/O field_6" at 237,236 size 96x32; FormatPattern 1
      ProcessValue <- "Logs2_DB_Display_Entry_ESD_Active"
   TextField "Text field_16" at 446,239 size 79x29; Text 'Avarie:'
   IOField "I/O field_7" at 527,239 size 96x32; FormatPattern 1
      ProcessValue <- "Logs2_DB_Display_Entry_Fault_Active"
   IOField "I/O field_11" at 309,120 size 304x32; FormatPattern 9999999999999999999999999999999999999999
      ProcessValue <- "Logs2_DB_Display_Entry_Timestamp"
   Button "Button_4" at 463,374 size 56x29; TextOff 'Gaseste'
      on Release: ResetBit("Logs2_DB_btn_latest")
      on Press: SetBit("Logs2_DB_btn_latest")
   TextField "Text field_17" at 361,378 size 98x20; Text 'Ultima intrare:'

screen "Logs3" 800x480
   TextField "Text field_1" at 23,455 size 60x20; Text 'Pompa 1'
   TextField "Text field_2" at 121,455 size 60x20; Text 'Pompa 2'
   TextField "Text field_3" at 221,455 size 60x20; Text 'Pompa 3'
   TextField "Text field_4" at 321,455 size 60x20; Text 'Pompa 4'
   TextField "Text field_5" at 429,455 size 43x20; Text 'Logs1'
   TextField "Text field_12" at 528,454 size 43x20; Text 'Logs2'
   TextField "Text field_14" at 627,453 size 43x20; Text 'Logs3'
   TextField "Text field_15" at 726,452 size 43x20; Text 'Logs4'
   TextField "Text field_11" at 357,3 size 68x27; Text 'Logs 3'
   TextField "Text field_6" at 552,65 size 98x20; Text 'Index Curent:'
   IOField "I/O field_1" at 647,63 size 29x25; FormatPattern 999
      ProcessValue <- "Logs3_DB_index"
   Button "Button_1" at 633,374 size 56x29; TextOff 'Inainte'
      on Release: ResetBit("Logs3_DB_btn_next")
      on Press: SetBit("Logs3_DB_btn_next")
   Button "Button_2" at 569,374 size 56x29; TextOff 'Inapoi'
      on Release: ResetBit("Logs3_DB_btn_prev")
      on Press: SetBit("Logs3_DB_btn_prev")
   TextField "Text field_7" at 127,377 size 88x20; Text 'Sari la index:'
   IOField "I/O field_2" at 220,375 size 29x25; FormatPattern 999
      ProcessValue <- "Logs3_DB_target_index"
   Button "Button_3" at 257,374 size 56x29; TextOff 'Gaseste'
      on Release: ResetBit("Logs3_DB_btn_jump")
      on Press: SetBit("Logs3_DB_btn_jump")
   TextField "Text field_8" at 177,176 size 65x29; Text 'Nivel:'
   IOField "I/O field_3" at 244,176 size 96x32; FormatPattern 999.99
      ProcessValue <- "Logs3_DB_Display_Entry_Level"
   TextField "Text field_9" at 446,179 size 58x29; Text 'Mod:'
   IOField "I/O field_4" at 510,179 size 96x32; FormatPattern 99
      ProcessValue <- "Logs3_DB_Display_Entry_Mode"
   TextField "Text field_10" at 175,120 size 130x29; Text 'Timestamp:'
   TextField "Text field_13" at 177,236 size 55x29; Text 'ESD:'
   IOField "I/O field_6" at 237,236 size 96x32; FormatPattern 1
      ProcessValue <- "Logs3_DB_Display_Entry_ESD_Active"
   TextField "Text field_16" at 446,239 size 79x29; Text 'Avarie:'
   IOField "I/O field_7" at 527,239 size 96x32; FormatPattern 1
      ProcessValue <- "Logs3_DB_Display_Entry_Fault_Active"
   IOField "I/O field_11" at 309,120 size 304x32; FormatPattern 9999999999999999999999999999999999999999
      ProcessValue <- "Logs3_DB_Display_Entry_Timestamp"
   Button "Button_4" at 463,374 size 56x29; TextOff 'Gaseste'
      on Release: ResetBit("Logs3_DB_btn_latest")
      on Press: SetBit("Logs3_DB_btn_latest")
   TextField "Text field_17" at 361,378 size 98x20; Text 'Ultima intrare:'

screen "Logs4" 800x480
   TextField "Text field_1" at 23,455 size 60x20; Text 'Pompa 1'
   TextField "Text field_2" at 121,455 size 60x20; Text 'Pompa 2'
   TextField "Text field_3" at 221,455 size 60x20; Text 'Pompa 3'
   TextField "Text field_4" at 321,455 size 60x20; Text 'Pompa 4'
   TextField "Text field_5" at 429,455 size 43x20; Text 'Logs1'
   TextField "Text field_12" at 528,454 size 43x20; Text 'Logs2'
   TextField "Text field_14" at 627,453 size 43x20; Text 'Logs3'
   TextField "Text field_15" at 726,452 size 43x20; Text 'Logs4'
   TextField "Text field_11" at 357,3 size 68x27; Text 'Logs 4'
   TextField "Text field_6" at 552,65 size 98x20; Text 'Index Curent:'
   IOField "I/O field_1" at 647,63 size 29x25; FormatPattern 999
      ProcessValue <- "Logs4_DB_index"
   Button "Button_1" at 633,374 size 56x29; TextOff 'Inainte'
      on Release: ResetBit("Logs4_DB_btn_next")
      on Press: SetBit("Logs4_DB_btn_next")
   Button "Button_2" at 569,374 size 56x29; TextOff 'Inapoi'
      on Release: ResetBit("Logs4_DB_btn_prev")
      on Press: SetBit("Logs4_DB_btn_prev")
   TextField "Text field_7" at 127,377 size 88x20; Text 'Sari la index:'
   IOField "I/O field_2" at 220,375 size 29x25; FormatPattern 999
      ProcessValue <- "Logs4_DB_target_index"
   Button "Button_3" at 257,374 size 56x29; TextOff 'Gaseste'
      on Release: ResetBit("Logs4_DB_btn_jump")
      on Press: SetBit("Logs4_DB_btn_jump")
   TextField "Text field_8" at 177,176 size 65x29; Text 'Nivel:'
   IOField "I/O field_3" at 244,176 size 96x32; FormatPattern 999.99
      ProcessValue <- "Logs4_DB_Display_Entry_Level"
   TextField "Text field_9" at 446,179 size 58x29; Text 'Mod:'
   IOField "I/O field_4" at 510,179 size 96x32; FormatPattern 99
      ProcessValue <- "Logs4_DB_Display_Entry_Mode"
   TextField "Text field_10" at 175,120 size 130x29; Text 'Timestamp:'
   TextField "Text field_13" at 177,236 size 55x29; Text 'ESD:'
   IOField "I/O field_6" at 237,236 size 96x32; FormatPattern 1
      ProcessValue <- "Logs4_DB_Display_Entry_ESD_Active"
   TextField "Text field_16" at 446,239 size 79x29; Text 'Avarie:'
   IOField "I/O field_7" at 527,239 size 96x32; FormatPattern 1
      ProcessValue <- "Logs4_DB_Display_Entry_Fault_Active"
   IOField "I/O field_11" at 309,120 size 304x32; FormatPattern 9999999999999999999999999999999999999999
      ProcessValue <- "Logs4_DB_Display_Entry_Timestamp"
   Button "Button_4" at 463,374 size 56x29; TextOff 'Gaseste'
      on Release: ResetBit("Logs4_DB_btn_latest")
      on Press: SetBit("Logs4_DB_btn_latest")
   TextField "Text field_17" at 361,378 size 98x20; Text 'Ultima intrare:'
*)